Universal Robots PolyScope program: PlaatsenHelicioDemostelling V3.4.1.urp

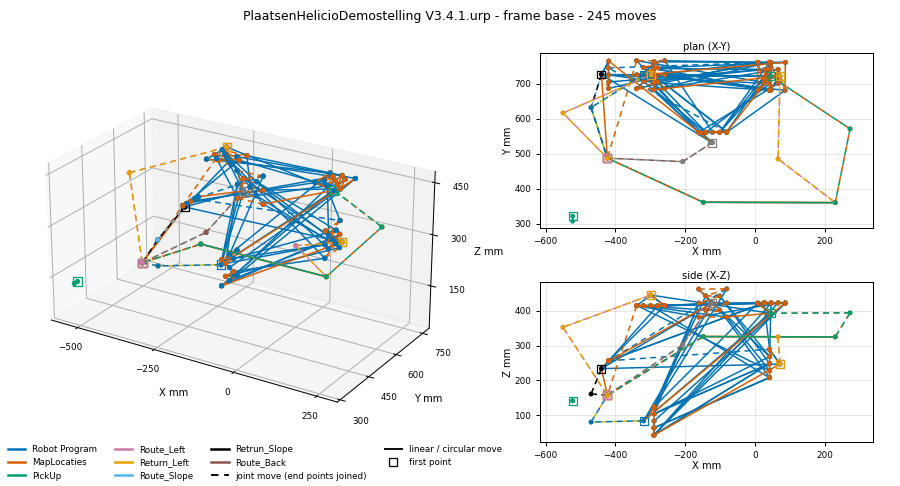
[picture p0: tool path of PlaatsenHelicioDemostelling V3.4.1.urp in frame base, 245 of 246 moves have a stored position in this frame; points joined in program order, loops and branches not executed]
Program PlaatsenHelicioDemostelling V3.4.1 (installation=TestOpstellingVDL directory=/programs/AA VDL ETG FvdT createdIn=5.13.0 lastSavedIn=5.13.0 robotSerialNumber=20195001449)
Calibrated DH parameters: a=[0.000035, -0.365107, -0.323271, 0.000053, -0.00002, 0]; d=[0.181019, -256.633431, 683.600492, -426.792497, 0.119803, 0.115725]; alpha=[1.570596, 0.001914, 0.001103, 1.570723, -1.571951, 0]; deltaTheta=[0, -0.931514, 8.183833, -0.969128, 0.000002, 0]
InitVariablesNode
BeforeStart
  Script file /programs/AA VDL ETG FvdT/Inspectie.script
    | ###
    | # Next functions are for the inspection how deep the helicoils are placed inside their holes ;)
    | # DirectiomalMovement is a variable that will tell the fucntion what axis is used for the movement:
    | # 0: X
    | # 1: Y
    | # 2: Z
    | # 3: XZ
    | ###
    | 
    | 
    | #Arrays to inspect the placed helicoils
    | global arrayStartX        = [0,0,0,0,0,0]
    | global arrayStartZ        = [0,0,0,0,0,0]
    | global arrayFinishX       = [0,0,0,0,0,0]
    | global arrayFinishZ       = [0,0,0,0,0,0]
    | #Results from the inspection
    | global ControlShort      = [0,0,0,0,0,0]
    | global ControlLong       = [0,0,0,0,0,0]
    | global ControlSpecial    = [0,0,0,0,0,0]
    | global ControlWrong      = [0,0,0,0,0,0]
    | global ControlSingle     = [0,0,0,0,0,0]
    | 
    | #How many went wrong while placing helicoils
    | global Interventions     = 0
    | 
    | #When calling this function it will return the wanted XYZ pose from the tcp
    | def Postion(RouteIndex, Start, PostionArrayX,PostionArrayZ):
    |   arrayX = PostionArrayX
    |   arrayZ = PostionArrayZ
    |   freedrive_mode()
    |   sleep(0.01)
    |   Pose  = get_actual_tcp_pose()
    |   end_freedrive_mode()
    |   sleep(0.01)
    |   arrayX[RouteIndex] = Pose[0]
    |   arrayZ[RouteIndex] = Pose[2]
    |   if (Start):
    |     arrayStartX = arrayX
    |     arrayStartZ = arrayZ
    |   else:
    |     arrayFinishX = arrayX
    |     arrayFinishZ = arrayZ
    |   end
    | end
    | 
    | #This function is for checking if the helicoil is placed at the right height everything is in mm. only the postionArrays are in meters
    | # 0: Right
    | # 1: Left
    | # 2: Slope
    | # 3: Back
    | # 4: Flat
    | # 5: Upside
    | def PostionControl(RouteIndex, Side, Route ,ToolcollarDistance, ControlArray):
    | array= ControlArray
    | if Side == 0:
    |   array[RouteIndex] = arrayStartX[RouteIndex] - arrayFinishX[RouteIndex]
    | elif Side == 1:
    |   array[RouteIndex] = arrayStartX[RouteIndex] - arrayFinishX[RouteIndex]
    | elif Side == 2:
    |   xstart = arrayStartX[RouteIndex]/-1
    |   xend = arrayFinishX[RouteIndex]/-1
    |   x = xstart - xend
    |   zstart = arrayStartZ[RouteIndex]
    |   zend   = arrayFinishZ[RouteIndex]
    |   z = zend - zstart
    |   x2 = x*x
    |   z2 = z*z
    |   result= x2+z2
    |   square = sqrt(result)
    |   mmSquare = square * 1000
    |   array[RouteIndex] = mmSquare - 1.5 - ToolcollarDistance
    | elif Side == 3:
    |   array[RouteIndex] = arrayStartX[RouteIndex] - arrayFinishX[RouteIndex]
    | elif Side == 4:
    |   array[RouteIndex] = arrayStartX[RouteIndex] - arrayFinishX[RouteIndex]
    | elif Side == 5:
    |   array[RouteIndex] = arrayStartX[RouteIndex] - arrayFinishX[RouteIndex]
    | end
    | 
    | if Route == 0:
    |   ControlShort = array
    | elif Route == 1:
    |   ControlSpecial = array
    | elif Route == 2:
    |   ControlSingle = array
    | elif Route == 3:
    |   ControlLong = array
    | elif Route == 4:
    |   ControlWrong = array
    | end
    |   if ((array[RouteIndex] < 0.1) and (array[RouteIndex] > 0.3)):
    |     popup("Helicoil outside the correct range of placement", title="Popup", warning=False, error=True)
    |     Interventions = Interventions + 1
    |   end
    | end
  Set DigitalOutput pin=digital_out[6]; digitalValue=1
  bFreedrive := 0
  bIndraaien := 0
  bOppakken := 0
  bUitdraaien := 0
  Route_Index_1 := 0
  URCap Move Shank (OnRobot, OnRobot A/S) dataModel(or-initialized=true, sd-target-pos=0.0)
    'Add conditions here'
Robot Program (runOnlyOnce=false)
  Route_Index_1 := 0
  Wait Condition expression=digital_in[0] or digital_in[1] or digital_in[2] or digital_in[3] or digital_in[4]
  If digital_in[0] and (ChoiceLong≟0)
    Folder LongDemo_1
      SafeHome (positionOptionType=SPEED_AND_ACCELERATION speed=1.047198 acceleration=1.396263 nextMotionTime=2)
      Call PickUp
      Call Route_Left
      MoveL speed 250 mm/s, acceleration 1200 mm/s^2 (useActiveTCP=true) feature=Base
        Waypoint App_Left: TCP in base x=71.596 y=722.403 z=247.152 mm, rx=1.2411 ry=-1.1842 rz=-1.247 rad; joints [84.654, -103.11, -124.444, -129.739, -95.317, 0.645] deg; TCP offset x=153 y=0 z=95.6 mm, rx=0 ry=1.5708 rz=0 rad
      MoveL speed 250 mm/s, acceleration 1200 mm/s^2 (useActiveTCP=true) feature=Center_Left
        Waypoint Left_Hole_1: TCP in base x=41.747 y=681.929 z=288.064 mm, rx=1.241 ry=-1.1844 rz=-1.2467 rad; joints [87.736, -95.501, -128.056, -133.774, -92.257, 0.486] deg; feature pose in base x=41.627 y=722.371 z=247.13 mm, rx=1.2411 ry=-1.1843 rz=-1.2469 rad
      Call ScrewIn_Left
      Call ScrewOut_Left
      Script: PostionControl(Route_Index_1,1, 3,20.4,ControlLong)
      Route_Index_1 := Route_Index_1+1
      MoveL speed 250 mm/s, acceleration 1200 mm/s^2 (useActiveTCP=true) feature=Center_Left
        Waypoint Left_Hole_1: TCP in base x=41.747 y=681.929 z=288.064 mm, rx=1.241 ry=-1.1844 rz=-1.2467 rad; joints [87.736, -95.501, -128.056, -133.774, -92.257, 0.486] deg
      MoveL speed 250 mm/s, acceleration 1200 mm/s^2 (useActiveTCP=true) feature=Base
        Waypoint App_Left: TCP in base x=71.596 y=722.403 z=247.152 mm, rx=1.2411 ry=-1.1842 rz=-1.247 rad; joints [84.654, -103.11, -124.444, -129.739, -95.317, 0.645] deg
      Call Return_Left
      Call PickUp
      Call Route_Slope
      MoveL speed 250 mm/s, acceleration 1200 mm/s^2 (useActiveTCP=true) feature=Base
        Waypoint App_Slope: TCP in base x=-439.97 y=727.052 z=233.948 mm, rx=-1.2131 ry=0.0047 rz=-2.8458 rad; joints [144.347, -130.504, -80.638, -95.321, 64.034, 60.975] deg
      MoveL speed 250 mm/s, acceleration 1200 mm/s^2 (useActiveTCP=true) feature=Center_Slope
        Waypoint Slope_Hole_1: TCP in base x=-418.988 y=765.455 z=256.032 mm, rx=-1.2134 ry=0.0048 rz=-2.8459 rad; joints [141.834, -130.588, -78.129, -96.713, 62.566, 58.706] deg; feature pose in base x=-417.692 y=727.543 z=255.471 mm, rx=-1.2135 ry=0.0049 rz=-2.8456 rad
      Call ScrewIn_Slope
      Call ScrewOut_Slope
      Script: PostionControl(Route_Index_1,2, 3,20.4,ControlLong)
      Route_Index_1 := Route_Index_1+1
      MoveL speed 250 mm/s, acceleration 1200 mm/s^2 (useActiveTCP=true) feature=Center_Slope
        Waypoint Slope_Hole_1: TCP in base x=-418.988 y=765.455 z=256.032 mm, rx=-1.2134 ry=0.0048 rz=-2.8459 rad; joints [141.834, -130.588, -78.129, -96.713, 62.566, 58.706] deg
      MoveL speed 250 mm/s, acceleration 1200 mm/s^2 (useActiveTCP=true) feature=Base
        Waypoint App_Slope: TCP in base x=-439.97 y=727.052 z=233.948 mm, rx=-1.2131 ry=0.0047 rz=-2.8458 rad; joints [144.347, -130.504, -80.638, -95.321, 64.034, 60.975] deg
      Call Retrun_Slope
      Call PickUp
      Call Route_Back
      MoveL speed 250 mm/s, acceleration 1200 mm/s^2 (useActiveTCP=true) feature=Base
        Waypoint App_Back: TCP in base x=-123.1 y=531.725 z=421.395 mm, rx=-1.1912 ry=-1.1756 rz=-1.1726 rad; joints [133.279, -56.474, -130.364, -80.605, 90.835, -48.335] deg
      MoveL speed 250 mm/s, acceleration 1200 mm/s^2 (useActiveTCP=true) feature=Center_Back
        Waypoint Back_Hole_1: TCP in base x=-161.091 y=559.776 z=461.746 mm, rx=-1.1916 ry=-1.1754 rz=-1.1728 rad; joints [134.504, -60.988, -124.308, -82.128, 90.793, -47.089] deg; feature pose in base x=-123.174 y=561.721 z=421.393 mm, rx=-1.1912 ry=-1.1756 rz=-1.1725 rad
      Call ScrewIn_Back
      Call ScrewOut_Back
      Script: PostionControl(Route_Index_1,3, 3,20.4,ControlLong)
      Route_Index_1 := Route_Index_1+1
      MoveL speed 250 mm/s, acceleration 1200 mm/s^2 (useActiveTCP=true) feature=Center_Back
        Waypoint Back_Hole_1: TCP in base x=-161.091 y=559.776 z=461.746 mm, rx=-1.1916 ry=-1.1754 rz=-1.1728 rad; joints [134.504, -60.988, -124.308, -82.128, 90.793, -47.089] deg
      MoveL speed 250 mm/s, acceleration 1200 mm/s^2 (useActiveTCP=true) feature=Base
        Waypoint App_Back: TCP in base x=-123.1 y=531.725 z=421.395 mm, rx=-1.1912 ry=-1.1756 rz=-1.1726 rad; joints [133.279, -56.474, -130.364, -80.605, 90.835, -48.335] deg
      Call Return_Back
      Call PickUp
      Call Route_Right
      MoveL speed 250 mm/s, acceleration 1200 mm/s^2 (useActiveTCP=true) feature=Base
        Waypoint App_Right: TCP in base x=-319.122 y=726.35 z=84.615 mm, rx=-1.8156 ry=0.6848 rz=-1.8051 rad; joints [142.098, -124.495, -115.917, -1.496, 59.13, 44.861] deg; TCP offset x=153 y=0 z=95.6 mm, rx=0 ry=1.5708 rz=0 rad
      MoveL speed 250 mm/s, acceleration 1200 mm/s^2 (useActiveTCP=true) feature=Center_Right
        Waypoint Right_Hole_1: TCP in base x=-288.676 y=762.832 z=123.23 mm, rx=-1.6513 ry=0.8665 rz=-1.6389 rad; joints [140.517, -126.661, -116.023, 15.048, 50.947, 35.529] deg; TCP offset x=153 y=0 z=95.6 mm, rx=0 ry=1.5708 rz=0 rad; feature pose in base x=-289.14 y=726.341 z=83.917 mm, rx=-1.8154 ry=0.6847 rz=-1.8054 rad
      Call ScrewIn_Right
      Call ScrewOut_Right
      Script: PostionControl(Route_Index_1,0, 3,20.4,ControlLong)
      Route_Index_1 := Route_Index_1+1
      MoveL speed 250 mm/s, acceleration 1200 mm/s^2 (useActiveTCP=true) feature=Center_Right
        Waypoint Right_Hole_1: TCP in base x=-288.676 y=762.832 z=123.23 mm, rx=-1.6513 ry=0.8665 rz=-1.6389 rad; joints [140.517, -126.661, -116.023, 15.048, 50.947, 35.529] deg
      MoveL speed 250 mm/s, acceleration 1200 mm/s^2 (useActiveTCP=true) feature=Base
        Waypoint App_Right: TCP in base x=-319.122 y=726.35 z=84.615 mm, rx=-1.8156 ry=0.6848 rz=-1.8051 rad; joints [142.098, -124.495, -115.917, -1.496, 59.13, 44.861] deg; TCP offset x=153 y=0 z=95.6 mm, rx=0 ry=1.5708 rz=0 rad
      Call Retrun_Right
      Call PickUp
      Call Route_Upside
      MoveL speed 250 mm/s, acceleration 1200 mm/s^2 (useActiveTCP=true) feature=Base
        Waypoint App_Upside: TCP in base x=44.432 y=722.092 z=392.585 mm, rx=0.0098 ry=0.0116 rz=-1.5803 rad; joints [105.261, -99.805, -128.74, -130.763, -74.252, 90.052] deg; TCP offset x=153 y=0 z=95.6 mm, rx=0 ry=1.5708 rz=0 rad
      MoveL speed 250 mm/s, acceleration 1200 mm/s^2 (useActiveTCP=true) feature=Base
        Waypoint Upside_Hole_1: TCP in base x=7.793 y=681.564 z=421.754 mm, rx=0.0115 ry=0.0085 rz=-1.1224 rad; joints [99.071, -96.217, -128.805, -134.239, -106.684, 90.097] deg
      Call ScrewIn_Upside
      Call ScrewOut_Upside
      Script: PostionControl(Route_Index_1,5, 3,20.4,ControlLong)
      Route_Index_1 := Route_Index_1+1
      MoveL speed 250 mm/s, acceleration 1200 mm/s^2 (useActiveTCP=true) feature=Base
        Waypoint Upside_Hole_1: TCP in base x=7.793 y=681.564 z=421.754 mm, rx=0.0115 ry=0.0085 rz=-1.1224 rad; joints [99.071, -96.217, -128.805, -134.239, -106.684, 90.097] deg
      MoveL speed 250 mm/s, acceleration 1200 mm/s^2 (useActiveTCP=true) feature=Base
        Waypoint App_Upside: TCP in base x=44.432 y=722.092 z=392.585 mm, rx=0.0098 ry=0.0116 rz=-1.5803 rad; joints [105.261, -99.805, -128.74, -130.763, -74.252, 90.052] deg
      Call Return_Upside
      Call PickUp
      Call Route_Flat
      MoveL speed 250 mm/s, acceleration 1200 mm/s^2 (useActiveTCP=true) feature=Base
        Waypoint App_Flat: TCP in base x=-298.667 y=726.067 z=444.64 mm, rx=-0.093 ry=3.1337 rz=-0.0054 rad; joints [137.032, -122.864, -79.694, 22.109, -43.59, 90.001] deg
      MoveL speed 250 mm/s, acceleration 1200 mm/s^2 (useActiveTCP=true) feature=Center_Flat
        Waypoint Flat_Hole_1: TCP in base x=-259.128 y=686.324 z=414.438 mm, rx=-0.0932 ry=3.1334 rz=-0.006 rad; joints [137.195, -119.277, -88.838, 27.642, -43.744, 89.991] deg; feature pose in base x=-298.69 y=726.112 z=414.639 mm, rx=-0.0931 ry=3.1338 rz=-0.0052 rad
      Call ScrewIn_Flat
      Call ScrewOut_Flat
      Script: PostionControl(Route_Index_1,4, 3,20.4,ControlLong)
      Route_Index_1 := Route_Index_1+1
      MoveL speed 250 mm/s, acceleration 1200 mm/s^2 (useActiveTCP=true) feature=Center_Flat
        Waypoint Flat_Hole_1: TCP in base x=-259.128 y=686.324 z=414.438 mm, rx=-0.0932 ry=3.1334 rz=-0.006 rad; joints [137.195, -119.277, -88.838, 27.642, -43.744, 89.991] deg
      MoveL speed 250 mm/s, acceleration 1200 mm/s^2 (useActiveTCP=true) feature=Base
        Waypoint App_Flat: TCP in base x=-298.667 y=726.067 z=444.64 mm, rx=-0.093 ry=3.1337 rz=-0.0054 rad; joints [137.032, -122.864, -79.694, 22.109, -43.59, 90.001] deg
      Call Return_Flat
      ChoiceLong := ChoiceLong+1
  ElseIf digital_in[0] and (ChoiceLong>1)
    Set DigitalOutput pin=digital_out[2]; digitalValue=1
    Wait Sleep waitTime=0.5
    Wait DigitalInput pin=digital_in[0]; digitalValue=1
    Set DigitalOutput pin=digital_out[2]; digitalValue=0
    Wait Sleep waitTime=0.5
  ElseIf digital_in[0] and (ChoiceLong≟1)
    Folder LongDemo2
      SafeHome (positionOptionType=SPEED_AND_ACCELERATION speed=1.047198 acceleration=1.396263 nextMotionTime=2)
      Call PickUp
      Call Route_Flat
      MoveL speed 250 mm/s, acceleration 1200 mm/s^2 (useActiveTCP=true) feature=Center_Flat
        Waypoint Flat_Hole_2: TCP in base x=-339.559 y=686.213 z=413.913 mm, rx=-0.0931 ry=3.1333 rz=-0.0061 rad; joints [140.84, -123.458, -82.105, 25.101, -47.4, 89.95] deg; feature pose in base x=-298.69 y=726.112 z=414.639 mm, rx=-0.0931 ry=3.1338 rz=-0.0052 rad
      Call ScrewIn_Flat
      Call ScrewOut_Flat
      Script: PostionControl(Route_Index_1,4, 3,20.4,ControlLong)
      Route_Index_1 := Route_Index_1+1
      MoveL speed 250 mm/s, acceleration 1200 mm/s^2 (useActiveTCP=true) feature=Center_Flat
        Waypoint Flat_Hole_2: TCP in base x=-339.559 y=686.213 z=413.913 mm, rx=-0.0931 ry=3.1333 rz=-0.0061 rad; joints [140.84, -123.458, -82.105, 25.101, -47.4, 89.95] deg
      Call Return_Flat
      Call PickUp
      Call Route_Upside
      MoveL speed 250 mm/s, acceleration 1200 mm/s^2 (useActiveTCP=true) feature=Base
        Waypoint Upside_Hole_2: TCP in base x=7.992 y=762.089 z=421.467 mm, rx=0.0114 ry=0.0085 rz=-1.1226 rad; joints [97.734, -103.064, -120.286, -135.906, -108.002, 90.119] deg
      Call ScrewIn_Upside
      Call ScrewOut_Upside
      Script: PostionControl(Route_Index_1,5, 3,20.4,ControlLong)
      Route_Index_1 := Route_Index_1+1
      MoveL speed 250 mm/s, acceleration 1200 mm/s^2 (useActiveTCP=true) feature=Base
        Waypoint Upside_Hole_2: TCP in base x=7.992 y=762.089 z=421.467 mm, rx=0.0114 ry=0.0085 rz=-1.1226 rad; joints [97.734, -103.064, -120.286, -135.906, -108.002, 90.119] deg
      Call Return_Upside
      Call PickUp
      Call Route_Right
      MoveL speed 250 mm/s, acceleration 1200 mm/s^2 (useActiveTCP=true) feature=Center_Right
        Waypoint Right_Hole_2: TCP in base x=-288.899 y=724.109 z=124.718 mm, rx=-1.8156 ry=0.6847 rz=-1.8052 rad; joints [140.747, -119.909, -118.016, -3.275, 59.778, 43.466] deg; feature pose in base x=-289.14 y=726.341 z=83.917 mm, rx=-1.8154 ry=0.6847 rz=-1.8054 rad
      Call ScrewIn_Right
      Call ScrewOut_Right
      Script: PostionControl(Route_Index_1,0, 3,20.4,ControlLong)
      Route_Index_1 := Route_Index_1+1
      MoveL speed 250 mm/s, acceleration 1200 mm/s^2 (useActiveTCP=true) feature=Center_Right
        Waypoint Right_Hole_2: TCP in base x=-288.899 y=724.109 z=124.718 mm, rx=-1.8156 ry=0.6847 rz=-1.8052 rad; joints [140.747, -119.909, -118.016, -3.275, 59.778, 43.466] deg
      Call Retrun_Right
      Call PickUp
      Call Route_Back
      MoveL speed 250 mm/s, acceleration 1200 mm/s^2 (useActiveTCP=true) feature=Center_Back
        Waypoint Back_Hole_2: TCP in base x=-81.106 y=561.818 z=462.255 mm, rx=-1.1915 ry=-1.1754 rz=-1.1728 rad; joints [125.05, -58.623, -125.311, -83.64, 91.187, -56.541] deg; feature pose in base x=-123.174 y=561.721 z=421.393 mm, rx=-1.1912 ry=-1.1756 rz=-1.1725 rad
      SuppressedNode
        Call ScrewIn_Back
      SuppressedNode
        Call ScrewOut_Back
      Script: PostionControl(Route_Index_1,3, 3,20.4,ControlLong)
      Route_Index_1 := Route_Index_1+1
      MoveL speed 250 mm/s, acceleration 1200 mm/s^2 (useActiveTCP=true) feature=Center_Back
        Waypoint Back_Hole_2: TCP in base x=-81.106 y=561.818 z=462.255 mm, rx=-1.1915 ry=-1.1754 rz=-1.1728 rad; joints [125.05, -58.623, -125.311, -83.64, 91.187, -56.541] deg
      Call Return_Back
      Call PickUp
      Call Route_Slope
      MoveJ speed 60 deg/s, acceleration 80 deg/s^2 (useActiveTCP=true) feature=Center_Slope
        Waypoint Slope_Hole_2: TCP in base x=-420.147 y=745.777 z=256.244 mm, rx=-1.2132 ry=0.0049 rz=-2.8457 rad; joints [142.781, -129.419, -80.121, -96.284, 63.105, 59.566] deg; feature pose in base x=-417.692 y=727.543 z=255.471 mm, rx=-1.2135 ry=0.0049 rz=-2.8456 rad
      Call ScrewIn_Slope
      Call ScrewOut_Slope
      Script: PostionControl(Route_Index_1,5, 3,20.4,ControlLong)
      Route_Index_1 := Route_Index_1+1
      MoveJ speed 60 deg/s, acceleration 80 deg/s^2 (useActiveTCP=true) feature=Center_Slope
        Waypoint Slope_Hole_2: TCP in base x=-420.147 y=745.777 z=256.244 mm, rx=-1.2132 ry=0.0049 rz=-2.8457 rad; joints [142.781, -129.419, -80.121, -96.284, 63.105, 59.566] deg
      Call Retrun_Slope
      Call PickUp
      Call Route_Left
      MoveJ speed 60 deg/s, acceleration 80 deg/s^2 (useActiveTCP=true) feature=Center_Left
        Waypoint Left_hole_2: TCP in base x=41.851 y=761.933 z=289.563 mm, rx=1.241 ry=-1.1846 rz=-1.2468 rad; joints [88.048, -101.94, -119.992, -135.397, -91.927, 0.472] deg; feature pose in base x=41.627 y=722.371 z=247.13 mm, rx=1.2411 ry=-1.1843 rz=-1.2469 rad
      Call ScrewIn_Left
      Call ScrewOut_Left
      Script: PostionControl(Route_Index_1,1, 3,20.4,ControlLong)
      Route_Index_1 := Route_Index_1+1
      MoveJ speed 60 deg/s, acceleration 80 deg/s^2 (useActiveTCP=true) feature=Center_Left
        Waypoint Left_hole_2: TCP in base x=41.851 y=761.933 z=289.563 mm, rx=1.241 ry=-1.1846 rz=-1.2468 rad; joints [88.048, -101.94, -119.992, -135.397, -91.927, 0.472] deg
      Call Return_Left
      ChoiceLong := ChoiceLong+1
  If digital_in[2] and (ChoiceSpecial≟0)
    Folder SpacialDemo_1
      SafeHome (positionOptionType=SPEED_AND_ACCELERATION speed=1.047198 acceleration=1.396263 nextMotionTime=2)
      Call PickUp
      Call Route_Upside
      MoveL speed 250 mm/s, acceleration 1200 mm/s^2 (useActiveTCP=true) feature=Base
        Waypoint Upside_Hole_3: TCP in base x=25.312 y=701.594 z=422.409 mm, rx=0.0095 ry=0.0108 rz=-1.6026 rad; joints [108.748, -95.233, -129.852, -134.263, -69.496, 89.993] deg
      Call ScrewIn_Upside
      Call ScrewOut_Upside
      Script: PostionControl(Route_Index_1,5, 1,20.4,ControlSpecial)
      Route_Index_1 := Route_Index_1+1
      MoveL speed 250 mm/s, acceleration 1200 mm/s^2 (useActiveTCP=true) feature=Base
        Waypoint Upside_Hole_3: TCP in base x=25.312 y=701.594 z=422.409 mm, rx=0.0095 ry=0.0108 rz=-1.6026 rad; joints [108.748, -95.233, -129.852, -134.263, -69.496, 89.993] deg
      Call Return_Upside
      Call PickUp
      Call Route_Slope
      MoveL speed 250 mm/s, acceleration 1200 mm/s^2 (useActiveTCP=true) feature=Center_Slope
        Waypoint Slope_Hole_3: TCP in base x=-419.505 y=725.856 z=255.958 mm, rx=-1.2131 ry=0.0047 rz=-2.8457 rad; joints [143.7, -128.19, -82.264, -95.747, 63.645, 60.388] deg; feature pose in base x=-417.692 y=727.543 z=255.471 mm, rx=-1.2135 ry=0.0049 rz=-2.8456 rad
      Call ScrewIn_Slope
      Call ScrewOut_Slope
      Script: PostionControl(Route_Index_1,2, 1,20.4,ControlSpecial)
      Route_Index_1 := Route_Index_1+1
      MoveL speed 250 mm/s, acceleration 1200 mm/s^2 (useActiveTCP=true) feature=Center_Slope
        Waypoint Slope_Hole_3: TCP in base x=-419.505 y=725.856 z=255.958 mm, rx=-1.2131 ry=0.0047 rz=-2.8457 rad; joints [143.7, -128.19, -82.264, -95.747, 63.645, 60.388] deg
      Call Retrun_Slope
      Call PickUp
      Call Route_Flat
      MoveL speed 250 mm/s, acceleration 1200 mm/s^2 (useActiveTCP=true) feature=Center_Flat
        Waypoint Flat_Hole_3: TCP in base x=-279.053 y=706.316 z=414.093 mm, rx=-0.093 ry=3.1333 rz=-0.0061 rad; joints [137.112, -121.662, -85.035, 26.213, -43.671, 89.995] deg; feature pose in base x=-298.69 y=726.112 z=414.639 mm, rx=-0.0931 ry=3.1338 rz=-0.0052 rad
      Call ScrewIn_Flat
      Call ScrewOut_Left
      Script: PostionControl(Route_Index_1,1, 1,20.4,ControlSpecial)
      Route_Index_1 := Route_Index_1+1
      MoveL speed 250 mm/s, acceleration 1200 mm/s^2 (useActiveTCP=true) feature=Center_Flat
        Waypoint Flat_Hole_3: TCP in base x=-279.053 y=706.316 z=414.093 mm, rx=-0.093 ry=3.1333 rz=-0.0061 rad; joints [137.112, -121.662, -85.035, 26.213, -43.671, 89.995] deg
      Call Return_Flat
      ChoiceSpecial := ChoiceSpecial+1
  ElseIf digital_in[2] and (ChoiceSpecial≟1)
    Folder SpacialDemo_2
      SafeHome (positionOptionType=SPEED_AND_ACCELERATION speed=1.047198 acceleration=1.396263 nextMotionTime=2)
      Call PickUp
      Call Route_Flat
      MoveL speed 250 mm/s, acceleration 1200 mm/s^2 (useActiveTCP=true) feature=Center_Flat
        Waypoint Flat_Hole_4: TCP in base x=-319.374 y=706.548 z=413.961 mm, rx=-0.093 ry=3.1333 rz=-0.0061 rad; joints [138.927, -123.752, -81.611, 24.894, -45.487, 89.973] deg
      Call ScrewIn_Flat
      Call ScrewOut_Flat
      Script: PostionControl(Route_Index_1,4, 1,20.4,ControlSpecial)
      Route_Index_1 := Route_Index_1+1
      MoveL speed 250 mm/s, acceleration 1200 mm/s^2 (useActiveTCP=true) feature=Center_Flat
        Waypoint Flat_Hole_4: TCP in base x=-319.374 y=706.548 z=413.961 mm, rx=-0.093 ry=3.1333 rz=-0.0061 rad; joints [138.927, -123.752, -81.611, 24.894, -45.487, 89.973] deg
      Call Return_Flat
      Call PickUp
      Call Route_Upside
      MoveL speed 250 mm/s, acceleration 1200 mm/s^2 (useActiveTCP=true) feature=Base
        Waypoint Upside_Hole_4: TCP in base x=28.457 y=741.552 z=422.373 mm, rx=0.0116 ry=0.0086 rz=-1.1224 rad; joints [95.855, -101.646, -122.034, -135.547, -109.894, 90.144] deg
      Call ScrewIn_Upside
      Call ScrewOut_Upside
      Script: PostionControl(Route_Index_1,5, 1,20.4,ControlSpecial)
      Route_Index_1 := Route_Index_1+1
      MoveL speed 250 mm/s, acceleration 1200 mm/s^2 (useActiveTCP=true) feature=Base
        Waypoint Upside_Hole_4: TCP in base x=28.457 y=741.552 z=422.373 mm, rx=0.0116 ry=0.0086 rz=-1.1224 rad; joints [95.855, -101.646, -122.034, -135.547, -109.894, 90.144] deg
      Call Return_Upside
      Call PickUp
      Call Route_Slope
      MoveL speed 250 mm/s, acceleration 1200 mm/s^2 (useActiveTCP=true) feature=Center_Slope
        Waypoint Slope_Hole_4: TCP in base x=-418.797 y=705.709 z=257.194 mm, rx=-1.2136 ry=0.005 rz=-2.8455 rad; joints [144.651, -126.896, -84.317, -95.345, 64.216, 61.241] deg; feature pose in base x=-417.692 y=727.543 z=255.471 mm, rx=-1.2135 ry=0.0049 rz=-2.8456 rad
      Call ScrewIn_Slope
      Call ScrewOut_Slope
      Script: PostionControl(Route_Index_1,2, 1,20.4,ControlSpecial)
      Route_Index_1 := Route_Index_1+1
      MoveL speed 250 mm/s, acceleration 1200 mm/s^2 (useActiveTCP=true) feature=Center_Slope
        Waypoint Slope_Hole_4: TCP in base x=-418.797 y=705.709 z=257.194 mm, rx=-1.2136 ry=0.005 rz=-2.8455 rad; joints [144.651, -126.896, -84.317, -95.345, 64.216, 61.241] deg
      Call Retrun_Slope
      ChoiceSpecial := ChoiceSpecial+1
  ElseIf digital_in[2] and (ChoiceSpecial≟2)
    Folder SpacialDemo_3
      SafeHome (positionOptionType=SPEED_AND_ACCELERATION speed=1.047198 acceleration=1.396263 nextMotionTime=2)
      Call PickUp
      Call Route_Slope
      MoveL speed 250 mm/s, acceleration 1200 mm/s^2 (useActiveTCP=true) feature=Center_Slope
        Waypoint Slope_Hole_5: TCP in base x=-419.08 y=686.879 z=256.503 mm, rx=-1.2131 ry=0.0048 rz=-2.8457 rad; joints [145.6, -125.867, -86.129, -94.947, 64.778, 62.084] deg
      Call ScrewIn_Slope
      Call ScrewOut_Slope
      Script: PostionControl(Route_Index_1,2, 1,20.4,ControlSpecial)
      Route_Index_1 := Route_Index_1+1
      MoveL speed 250 mm/s, acceleration 1200 mm/s^2 (useActiveTCP=true) feature=Center_Slope
        Waypoint Slope_Hole_5: TCP in base x=-419.08 y=686.879 z=256.503 mm, rx=-1.2131 ry=0.0048 rz=-2.8457 rad; joints [145.6, -125.867, -86.129, -94.947, 64.778, 62.084] deg
      Call Retrun_Slope
      Call PickUp
      Call Route_Flat
      MoveL speed 250 mm/s, acceleration 1200 mm/s^2 (useActiveTCP=true) feature=Center_Flat
        Waypoint Flat_Hole_5: TCP in base x=-258.651 y=725.987 z=414.388 mm, rx=-0.0931 ry=3.1336 rz=-0.0055 rad; joints [135.168, -122.05, -84.362, 25.942, -41.726, 90.022] deg; feature pose in base x=-298.69 y=726.112 z=414.639 mm, rx=-0.0931 ry=3.1338 rz=-0.0052 rad
      Call ScrewIn_Flat
      Call ScrewOut_Flat
      Script: PostionControl(Route_Index_1,4, 1,20.4,ControlSpecial)
      Route_Index_1 := Route_Index_1+1
      MoveL speed 250 mm/s, acceleration 1200 mm/s^2 (useActiveTCP=true) feature=Center_Flat
        Waypoint Flat_Hole_5: TCP in base x=-258.651 y=725.987 z=414.388 mm, rx=-0.0931 ry=3.1336 rz=-0.0055 rad; joints [135.168, -122.05, -84.362, 25.942, -41.726, 90.022] deg
      Call Return_Flat
      Call PickUp
      Call Route_Upside
      MoveL speed 250 mm/s, acceleration 1200 mm/s^2 (useActiveTCP=true) feature=Base
        Waypoint Upside_Hole_5: TCP in base x=45.602 y=681.858 z=421.646 mm, rx=0.0094 ry=0.0108 rz=-1.5922 rad; joints [106.795, -93.58, -131.803, -133.972, -72.048, 90.021] deg
      SuppressedNode
        Call ScrewIn_Upside
      SuppressedNode
        Call ScrewOut_Upside
      Script: PostionControl(Route_Index_1,4, 1,20.5,ControlSpecial)
      MoveL speed 250 mm/s, acceleration 1200 mm/s^2 (useActiveTCP=true) feature=Base
        Waypoint Upside_Hole_5: TCP in base x=45.602 y=681.858 z=421.646 mm, rx=0.0094 ry=0.0108 rz=-1.5922 rad; joints [106.795, -93.58, -131.803, -133.972, -72.048, 90.021] deg
      Call Return_Upside
      ChoiceSpecial := ChoiceSpecial+1
  If digital_in[3] and (ChoiceWrong≟0)
    Folder WrongDemo_1
      SafeHome (positionOptionType=SPEED_AND_ACCELERATION speed=1.047198 acceleration=1.396263 nextMotionTime=2)
      Call PickUp
      Call Route_Left
      MoveL speed 250 mm/s, acceleration 1200 mm/s^2 (useActiveTCP=true) feature=Center_Left
        Waypoint Left_Hole_3: TCP in base x=41.78 y=700.693 z=268.277 mm, rx=1.2407 ry=-1.1848 rz=-1.2467 rad; joints [87.825, -98.689, -127.06, -131.593, -92.143, 0.481] deg; feature pose in base x=41.627 y=722.371 z=247.13 mm, rx=1.2411 ry=-1.1843 rz=-1.2469 rad
      Call ScrewIn_Left
      Call ScrewOut_Left
      Script: PostionControl(Route_Index_1,1, 4,20.4,ControlWrong)
      Route_Index_1 := Route_Index_1+1
      MoveL speed 250 mm/s, acceleration 1200 mm/s^2 (useActiveTCP=true) feature=Center_Left
        Waypoint Left_Hole_3: TCP in base x=41.78 y=700.693 z=268.277 mm, rx=1.2407 ry=-1.1848 rz=-1.2467 rad; joints [87.825, -98.689, -127.06, -131.593, -92.143, 0.481] deg
      Call Return_Left
      Call PickUp
      Call Route_Back
      MoveL speed 250 mm/s, acceleration 1200 mm/s^2 (useActiveTCP=true) feature=Center_Back
        Waypoint Back_Hole_3: TCP in base x=-141.317 y=560.737 z=442.316 mm, rx=-1.1916 ry=-1.1753 rz=-1.1725 rad; joints [132.279, -60.529, -126.481, -80.438, 90.901, -49.317] deg; feature pose in base x=-123.174 y=561.721 z=421.393 mm, rx=-1.1912 ry=-1.1756 rz=-1.1725 rad
      Call ScrewIn_Back
      Call ScrewOut_Back
      Script: PostionControl(Route_Index_1,1, 3,20.4,ControlWrong)
      Route_Index_1 := Route_Index_1+1
      MoveL speed 250 mm/s, acceleration 1200 mm/s^2 (useActiveTCP=true) feature=Center_Back
        Waypoint Back_Hole_3: TCP in base x=-141.317 y=560.737 z=442.316 mm, rx=-1.1916 ry=-1.1753 rz=-1.1725 rad; joints [132.279, -60.529, -126.481, -80.438, 90.901, -49.317] deg
      Call Return_Back
      Call PickUp
      Call Route_Right
      MoveL speed 250 mm/s, acceleration 1200 mm/s^2 (useActiveTCP=true) feature=Center_Right
        Waypoint Right_Hole_3: TCP in base x=-289.204 y=683.885 z=123.717 mm, rx=-1.8156 ry=0.6847 rz=-1.8051 rad; joints [143.374, -117.868, -121.795, -2.924, 58.544, 46.159] deg; feature pose in base x=-289.14 y=726.341 z=83.917 mm, rx=-1.8154 ry=0.6847 rz=-1.8054 rad
      Call ScrewIn_Right
      Call ScrewOut_Right
      Script: PostionControl(Route_Index_1,0, 4,20.4,ControlWrong)
      Route_Index_1 := Route_Index_1+1
      MoveL speed 250 mm/s, acceleration 1200 mm/s^2 (useActiveTCP=true) feature=Center_Right
        Waypoint Right_Hole_3: TCP in base x=-289.204 y=683.885 z=123.717 mm, rx=-1.8156 ry=0.6847 rz=-1.8051 rad; joints [143.374, -117.868, -121.795, -2.924, 58.544, 46.159] deg
      Call Retrun_Right
    ChoiceWrong := ChoiceWrong+1
  ElseIf digital_in[3] and (ChoiceWrong≟2)
    Folder WrongDemo_3
      SafeHome (positionOptionType=SPEED_AND_ACCELERATION speed=1.047198 acceleration=1.396263 nextMotionTime=2)
      Call PickUp
      Call Route_Back
      MoveL speed 250 mm/s, acceleration 1200 mm/s^2 (useActiveTCP=true) feature=Center_Back
        Waypoint Back_Hole_5: TCP in base x=-160.808 y=560.703 z=421.755 mm, rx=-1.1913 ry=-1.1757 rz=-1.1725 rad; joints [134.374, -61.689, -128.015, -77.73, 90.806, -47.239] deg; feature pose in base x=-123.174 y=561.721 z=421.393 mm, rx=-1.1912 ry=-1.1756 rz=-1.1725 rad
      Call ScrewIn_Back
      Call ScrewOut_Back
      Script: PostionControl(Route_Index_1,3, 4,20.4,ControlWrong)
      Route_Index_1 := Route_Index_1+1
      MoveL speed 250 mm/s, acceleration 1200 mm/s^2 (useActiveTCP=true) feature=Center_Back
        Waypoint Back_Hole_5: TCP in base x=-160.808 y=560.703 z=421.755 mm, rx=-1.1913 ry=-1.1757 rz=-1.1725 rad; joints [134.374, -61.689, -128.015, -77.73, 90.806, -47.239] deg
      Call Return_Back
      Call PickUp
      Call Route_Right
      MoveL speed 250 mm/s, acceleration 1200 mm/s^2 (useActiveTCP=true) feature=Center_Right
        Waypoint Right_Hole_5: TCP in base x=-289.172 y=703.708 z=104.449 mm, rx=-1.8156 ry=0.6847 rz=-1.8052 rad; joints [142.057, -120.721, -120.085, -1.08, 59.155, 44.81] deg; feature pose in base x=-289.14 y=726.341 z=83.917 mm, rx=-1.8154 ry=0.6847 rz=-1.8054 rad
      Call ScrewIn_Right
      Call ScrewOut_Right
      Script: PostionControl(Route_Index_1,0, 4,20.4,ControlWrong)
      Route_Index_1 := Route_Index_1+1
      MoveL speed 250 mm/s, acceleration 1200 mm/s^2 (useActiveTCP=true) feature=Center_Right
        Waypoint Right_Hole_5: TCP in base x=-289.172 y=703.708 z=104.449 mm, rx=-1.8156 ry=0.6847 rz=-1.8052 rad; joints [142.057, -120.721, -120.085, -1.08, 59.155, 44.81] deg
      Call Retrun_Right
      Call PickUp
      Call Route_Left
      MoveL speed 250 mm/s, acceleration 1200 mm/s^2 (useActiveTCP=true) feature=Center_Left
        Waypoint Left_Hole_5: TCP in base x=41.621 y=681.741 z=247.936 mm, rx=1.2407 ry=-1.1848 rz=-1.2466 rad; joints [87.758, -98.951, -129.738, -128.658, -92.209, 0.483] deg; feature pose in base x=41.627 y=722.371 z=247.13 mm, rx=1.2411 ry=-1.1843 rz=-1.2469 rad
      Call ScrewIn_Left
      Call ScrewOut_Left
      Script: PostionControl(Route_Index_1,1, 4,20.4,ControlWrong)
      Route_Index_1 := Route_Index_1+1
      MoveL speed 250 mm/s, acceleration 1200 mm/s^2 (useActiveTCP=true) feature=Center_Left
        Waypoint Left_Hole_5: TCP in base x=41.621 y=681.741 z=247.936 mm, rx=1.2407 ry=-1.1848 rz=-1.2466 rad; joints [87.758, -98.951, -129.738, -128.658, -92.209, 0.483] deg
      Call Return_Left
    ChoiceWrong := ChoiceWrong+1
  ElseIf digital_in[3] and (ChoiceWrong≟1)
    Folder WrongDemo_2
      SafeHome (positionOptionType=SPEED_AND_ACCELERATION speed=1.047198 acceleration=1.396263 nextMotionTime=2)
      Call PickUp
      Call Route_Right
      MoveL speed 250 mm/s, acceleration 1200 mm/s^2 (useActiveTCP=true) feature=Center_Right
        Waypoint Right_Hole_4: TCP in base x=-288.818 y=744.018 z=104.467 mm, rx=-1.8156 ry=0.6845 rz=-1.8053 rad; joints [139.527, -122.763, -116.22, -1.612, 60.368, 42.243] deg; feature pose in base x=-289.14 y=726.341 z=83.917 mm, rx=-1.8154 ry=0.6847 rz=-1.8054 rad
      Call ScrewIn_Right
      Call ScrewOut_Right
      Script: PostionControl(Route_Index_1,0, 4,20.4,ControlWrong)
      Route_Index_1 := Route_Index_1+1
      MoveL speed 250 mm/s, acceleration 1200 mm/s^2 (useActiveTCP=true) feature=Center_Right
        Waypoint Right_Hole_4: TCP in base x=-288.818 y=744.018 z=104.467 mm, rx=-1.8156 ry=0.6845 rz=-1.8053 rad; joints [139.527, -122.763, -116.22, -1.612, 60.368, 42.243] deg
      Call Retrun_Right
      Call PickUp
      Call Route_Left
      MoveL speed 250 mm/s, acceleration 1200 mm/s^2 (useActiveTCP=true) feature=Center_Left
        Waypoint Left_Hole_4: TCP in base x=41.829 y=741.625 z=268.564 mm, rx=1.2407 ry=-1.1848 rz=-1.2468 rad; joints [87.983, -101.916, -122.916, -132.511, -91.98, 0.478] deg; feature pose in base x=41.627 y=722.371 z=247.13 mm, rx=1.2411 ry=-1.1843 rz=-1.2469 rad
      Call ScrewIn_Left
      Call ScrewOut_Left
      Script: PostionControl(Route_Index_1,1, 4,20.4,ControlWrong)
      Route_Index_1 := Route_Index_1+1
      MoveL speed 250 mm/s, acceleration 1200 mm/s^2 (useActiveTCP=true) feature=Center_Left
        Waypoint Left_Hole_4: TCP in base x=41.829 y=741.625 z=268.564 mm, rx=1.2407 ry=-1.1848 rz=-1.2468 rad; joints [87.983, -101.916, -122.916, -132.511, -91.98, 0.478] deg
      Call Return_Left
      Call PickUp
      Call Route_Back
      MoveL speed 250 mm/s, acceleration 1200 mm/s^2 (useActiveTCP=true) feature=Center_Back
        Waypoint Back_Hole_4: TCP in base x=-100.931 y=561.75 z=441.913 mm, rx=-1.1915 ry=-1.1753 rz=-1.1725 rad; joints [127.507, -59.311, -127.065, -81.147, 91.1, -54.089] deg; feature pose in base x=-123.174 y=561.721 z=421.393 mm, rx=-1.1912 ry=-1.1756 rz=-1.1725 rad
      Call ScrewIn_Back
      Call ScrewOut_Back
      Script: PostionControl(Route_Index_1,3, 4,20.4,ControlWrong)
      Route_Index_1 := Route_Index_1+1
      MoveL speed 250 mm/s, acceleration 1200 mm/s^2 (useActiveTCP=true) feature=Center_Back
        Waypoint Back_Hole_4: TCP in base x=-100.931 y=561.75 z=441.913 mm, rx=-1.1915 ry=-1.1753 rz=-1.1725 rad; joints [127.507, -59.311, -127.065, -81.147, 91.1, -54.089] deg
      Call Return_Back
    ChoiceWrong := ChoiceWrong+1
  If digital_in[1] and (ChoiceShort≟0)
    Folder ShortDemo_1
      SafeHome (positionOptionType=SPEED_AND_ACCELERATION speed=1.047198 acceleration=1.396263 nextMotionTime=2)
      Call PickUp
      Call Route_Left
      MoveL speed 250 mm/s, acceleration 1200 mm/s^2 (useActiveTCP=true) feature=Center_Left
        Waypoint Left_Hole_6: TCP in base x=41.661 y=721.943 z=248.573 mm, rx=1.2412 ry=-1.1844 rz=-1.247 rad; joints [87.923, -102.032, -125.679, -129.603, -92.048, 0.482] deg; feature pose in base x=41.627 y=722.371 z=247.13 mm, rx=1.2411 ry=-1.1843 rz=-1.2469 rad
      Call ScrewIn_Left
      Call ScrewOut_Left
      Script: PostionControl(Route_Index_1,1, 0,20.4,ControlShort)
      Route_Index_1 := Route_Index_1+1
      MoveL speed 250 mm/s, acceleration 1200 mm/s^2 (useActiveTCP=true) feature=Center_Left
        Waypoint Left_Hole_6: TCP in base x=41.661 y=721.943 z=248.573 mm, rx=1.2412 ry=-1.1844 rz=-1.247 rad; joints [87.923, -102.032, -125.679, -129.603, -92.048, 0.482] deg
      Call Return_Left
      Call PickUp
      Call Route_Right
      MoveL speed 250 mm/s, acceleration 1200 mm/s^2 (useActiveTCP=true) feature=Center_Right
        Waypoint Right_Hole_10: TCP in base x=-289.595 y=723.359 z=43.588 mm, rx=-1.8156 ry=0.6846 rz=-1.8051 rad; joints [140.827, -127.475, -118.143, 4.367, 59.733, 43.565] deg; feature pose in base x=-289.14 y=726.341 z=83.917 mm, rx=-1.8154 ry=0.6847 rz=-1.8054 rad
      Call ScrewIn_Right
      Call ScrewOut_Right
      Script: PostionControl(Route_Index_1,0, 0,20.4,ControlShort)
      Route_Index_1 := Route_Index_1+1
      MoveL speed 250 mm/s, acceleration 1200 mm/s^2 (useActiveTCP=true) feature=Center_Right
        Waypoint Right_Hole_10: TCP in base x=-289.595 y=723.359 z=43.588 mm, rx=-1.8156 ry=0.6846 rz=-1.8051 rad; joints [140.827, -127.475, -118.143, 4.367, 59.733, 43.565] deg
      Call Retrun_Right
      Call PickUp
      Call Route_Upside
      MoveL speed 250 mm/s, acceleration 1200 mm/s^2 (useActiveTCP=true) feature=Base
        Waypoint Upside_Hole_6: TCP in base x=45.629 y=721.749 z=421.143 mm, rx=0.0098 ry=0.0115 rz=-1.5802 rad; joints [105.13, -97.306, -127.635, -134.374, -74.396, 90.048] deg
      Call ScrewIn_Upside
      Call ScrewOut_Upside
      Script: PostionControl(Route_Index_1,5, 0,20.4,ControlShort)
      Route_Index_1 := Route_Index_1+1
      MoveL speed 250 mm/s, acceleration 1200 mm/s^2 (useActiveTCP=true) feature=Base
        Waypoint Upside_Hole_6: TCP in base x=45.629 y=721.749 z=421.143 mm, rx=0.0098 ry=0.0115 rz=-1.5802 rad; joints [105.13, -97.306, -127.635, -134.374, -74.396, 90.048] deg
      Call Return_Upside
    ChoiceShort := ChoiceShort+1
  ElseIf digital_in[1] and (ChoiceShort≟1)
    Folder ShortDemo_2
      SafeHome (positionOptionType=SPEED_AND_ACCELERATION speed=1.047198 acceleration=1.396263 nextMotionTime=2)
      Call PickUp
      Call Route_Upside
      MoveL speed 250 mm/s, acceleration 1200 mm/s^2 (useActiveTCP=true) feature=Base
        Waypoint Upside_Hole_7: TCP in base x=46.075 y=761.507 z=422.684 mm, rx=0.0095 ry=0.0109 rz=-1.5923 rad; joints [104.212, -100.607, -123.332, -135.408, -74.616, 90.054] deg
      Call ScrewIn_Upside
      Call ScrewOut_Upside
      Script: PostionControl(Route_Index_1,5, 0,20.4,ControlShort)
      Route_Index_1 := Route_Index_1+1
      MoveL speed 250 mm/s, acceleration 1200 mm/s^2 (useActiveTCP=true) feature=Base
        Waypoint Upside_Hole_7: TCP in base x=46.075 y=761.507 z=422.684 mm, rx=0.0095 ry=0.0109 rz=-1.5923 rad; joints [104.212, -100.607, -123.332, -135.408, -74.616, 90.054] deg
      Call Return_Upside
      Call PickUp
      Call Route_Flat
      MoveL speed 250 mm/s, acceleration 1200 mm/s^2 (useActiveTCP=true) feature=Center_Flat
        Waypoint Flat_Hole_10: TCP in base x=-258.485 y=766.369 z=414.023 mm, rx=-0.0934 ry=3.1332 rz=-0.0063 rad; joints [133.268, -125.019, -79.495, 23.998, -39.818, 90.046] deg; feature pose in base x=-298.69 y=726.112 z=414.639 mm, rx=-0.0931 ry=3.1338 rz=-0.0052 rad
      Call ScrewIn_Flat
      Call ScrewOut_Flat
      Script: PostionControl(Route_Index_1,4, 0,20.4,ControlShort)
      Route_Index_1 := Route_Index_1+1
      MoveL speed 250 mm/s, acceleration 1200 mm/s^2 (useActiveTCP=true) feature=Center_Flat
        Waypoint Flat_Hole_10: TCP in base x=-258.485 y=766.369 z=414.023 mm, rx=-0.0934 ry=3.1332 rz=-0.0063 rad; joints [133.268, -125.019, -79.495, 23.998, -39.818, 90.046] deg
      Call Return_Flat
      Call PickUp
      Call Route_Back
      MoveL speed 250 mm/s, acceleration 1200 mm/s^2 (useActiveTCP=true) feature=Center_Back
        Waypoint Back_Hole_6: TCP in base x=-121.665 y=561.713 z=422.253 mm, rx=-1.1913 ry=-1.1757 rz=-1.1725 rad; joints [129.968, -60.258, -128.629, -78.606, 90.991, -51.642] deg; feature pose in base x=-123.174 y=561.721 z=421.393 mm, rx=-1.1912 ry=-1.1756 rz=-1.1725 rad
      Call ScrewIn_Back
      Call ScrewOut_Back
      Script: PostionControl(Route_Index_1,3, 0,20.4,ControlShort)
      Route_Index_1 := Route_Index_1+1
      MoveL speed 250 mm/s, acceleration 1200 mm/s^2 (useActiveTCP=true) feature=Center_Back
        Waypoint Back_Hole_6: TCP in base x=-121.665 y=561.713 z=422.253 mm, rx=-1.1913 ry=-1.1757 rz=-1.1725 rad; joints [129.968, -60.258, -128.629, -78.606, 90.991, -51.642] deg
      Call Return_Back
    ChoiceShort := ChoiceShort+1
  ElseIf digital_in[1] and (ChoiceShort≟2)
    Folder ShortDemo_3
      SafeHome (positionOptionType=SPEED_AND_ACCELERATION speed=1.047198 acceleration=1.396263 nextMotionTime=2)
      Call PickUp
      Call Route_Back
      MoveL speed 250 mm/s, acceleration 1200 mm/s^2 (useActiveTCP=true) feature=Center_Back
        Waypoint Back_Hole_7: TCP in base x=-81.214 y=561.376 z=422.087 mm, rx=-1.1914 ry=-1.1756 rz=-1.1725 rad; joints [125.096, -59.068, -129.167, -79.339, 91.196, -56.509] deg
      Call ScrewIn_Back
      Call ScrewOut_Back
      Script: PostionControl(Route_Index_1,3, 0,20.4,ControlShort)
      Route_Index_1 := Route_Index_1+1
      MoveL speed 250 mm/s, acceleration 1200 mm/s^2 (useActiveTCP=true) feature=Center_Back
        Waypoint Back_Hole_7: TCP in base x=-81.214 y=561.376 z=422.087 mm, rx=-1.1914 ry=-1.1756 rz=-1.1725 rad; joints [125.096, -59.068, -129.167, -79.339, 91.196, -56.509] deg
      Call Return_Back
      Call PickUp
      Call Route_Upside
      MoveL speed 250 mm/s, acceleration 1200 mm/s^2 (useActiveTCP=true) feature=Base
        Waypoint Upside_Hole_10: TCP in base x=85.909 y=681.545 z=420.624 mm, rx=0.0097 ry=0.0115 rz=-1.58 rad; joints [101.434, -94.182, -131.306, -133.827, -78.105, 90.095] deg
      Call ScrewIn_Upside
      Call ScrewOut_Upside
      Script: PostionControl(Route_Index_1,5, 0,20.4,ControlShort)
      Route_Index_1 := Route_Index_1+1
      MoveL speed 250 mm/s, acceleration 1200 mm/s^2 (useActiveTCP=true) feature=Base
        Waypoint Upside_Hole_10: TCP in base x=85.909 y=681.545 z=420.624 mm, rx=0.0097 ry=0.0115 rz=-1.58 rad; joints [101.434, -94.182, -131.306, -133.827, -78.105, 90.095] deg
      Call Return_Upside
      Call PickUp
      Call Route_Right
      MoveL speed 250 mm/s, acceleration 1200 mm/s^2 (useActiveTCP=true) feature=Center_Right
        Waypoint Right_Hole_6: TCP in base x=-289.189 y=724.036 z=83.936 mm, rx=-1.8154 ry=0.6846 rz=-1.8053 rad; joints [140.767, -123.659, -118.205, 0.642, 59.757, 43.494] deg; feature pose in base x=-289.14 y=726.341 z=83.917 mm, rx=-1.8154 ry=0.6847 rz=-1.8054 rad
      Call ScrewIn_Right
      Call ScrewOut_Right
      Script: PostionControl(Route_Index_1,0, 0,20.4,ControlShort)
      Route_Index_1 := Route_Index_1+1
      MoveL speed 250 mm/s, acceleration 1200 mm/s^2 (useActiveTCP=true) feature=Center_Right
        Waypoint Right_Hole_6: TCP in base x=-289.189 y=724.036 z=83.936 mm, rx=-1.8154 ry=0.6846 rz=-1.8053 rad; joints [140.767, -123.659, -118.205, 0.642, 59.757, 43.494] deg
      Call Retrun_Right
    ChoiceShort := ChoiceShort+1
  ElseIf digital_in[1] and (ChoiceShort≟3)
    Folder ShortDemo_4
      SafeHome (positionOptionType=SPEED_AND_ACCELERATION speed=1.047198 acceleration=1.396263 nextMotionTime=2)
      Call PickUp
      Call Route_Right
      MoveL speed 250 mm/s, acceleration 1200 mm/s^2 (useActiveTCP=true) feature=Center_Right
        Waypoint Right_Hole_7: TCP in base x=-289.188 y=743.625 z=64.091 mm, rx=-1.8156 ry=0.6847 rz=-1.8052 rad; joints [139.569, -126.432, -116.277, 2.096, 60.342, 42.295] deg
      Call ScrewIn_Right
      Call ScrewOut_Right
      Wait Sleep waitTime=10
      SuppressedNode
        Script: PostionControl(Route_Index_1,0, 0,20.4,ControlShort)
      Route_Index_1 := Route_Index_1+1
      MoveL speed 250 mm/s, acceleration 1200 mm/s^2 (useActiveTCP=true) feature=Center_Right
        Waypoint Right_Hole_7: TCP in base x=-289.188 y=743.625 z=64.091 mm, rx=-1.8156 ry=0.6847 rz=-1.8052 rad; joints [139.569, -126.432, -116.277, 2.096, 60.342, 42.295] deg
      Call Retrun_Right
      Call PickUp
      Call Route_Left
      MoveL speed 250 mm/s, acceleration 1200 mm/s^2 (useActiveTCP=true) feature=Center_Left
        Waypoint Left_Hole_10: TCP in base x=41.475 y=682.374 z=207.743 mm, rx=1.2403 ry=-1.1849 rz=-1.2465 rad; joints [87.783, -102.844, -131.026, -123.494, -92.168, 0.493] deg; feature pose in base x=41.627 y=722.371 z=247.13 mm, rx=1.2411 ry=-1.1843 rz=-1.2469 rad
      Call ScrewIn_Left
      Call ScrewOut_Left
      Script: PostionControl(Route_Index_1,1, 0,20.4,ControlShort)
      Route_Index_1 := Route_Index_1+1
      MoveL speed 250 mm/s, acceleration 1200 mm/s^2 (useActiveTCP=true) feature=Center_Left
        Waypoint Left_Hole_10: TCP in base x=41.475 y=682.374 z=207.743 mm, rx=1.2403 ry=-1.1849 rz=-1.2465 rad; joints [87.783, -102.844, -131.026, -123.494, -92.168, 0.493] deg
      Call Return_Left
      Call PickUp
      Call Route_Flat
      MoveL speed 250 mm/s, acceleration 1200 mm/s^2 (useActiveTCP=true) feature=Center_Flat
        Waypoint Flat_Hole_6: TCP in base x=-298.708 y=726.085 z=414.645 mm, rx=-0.0931 ry=3.1337 rz=-0.0053 rad; joints [137.035, -124.015, -81.089, 24.659, -43.595, 90] deg; feature pose in base x=-298.69 y=726.112 z=414.639 mm, rx=-0.0931 ry=3.1338 rz=-0.0052 rad
      Call ScrewIn_Flat
      Wait Sleep waitTime=1
      Call ScrewOut_Flat
      Wait Sleep waitTime=20
      Script: PostionControl(Route_Index_1,4, 0,20.4,ControlShort)
      Route_Index_1 := Route_Index_1+1
      MoveL speed 250 mm/s, acceleration 1200 mm/s^2 (useActiveTCP=true) feature=Center_Flat
        Waypoint Flat_Hole_6: TCP in base x=-298.708 y=726.085 z=414.645 mm, rx=-0.0931 ry=3.1337 rz=-0.0053 rad; joints [137.035, -124.015, -81.089, 24.659, -43.595, 90] deg
      Call Return_Flat
    ChoiceShort := ChoiceShort+1
  ElseIf digital_in[1] and (ChoiceShort≟4)
    Folder ShortDemo_5
      SafeHome (positionOptionType=SPEED_AND_ACCELERATION speed=1.047198 acceleration=1.396263 nextMotionTime=2)
      Call PickUp
      Call Route_Flat
      MoveL speed 250 mm/s, acceleration 1200 mm/s^2 (useActiveTCP=true) feature=Center_Flat
        Waypoint Flat_Hole_7: TCP in base x=-338.996 y=726.099 z=413.978 mm, rx=-0.093 ry=3.1337 rz=-0.0056 rad; joints [138.802, -126.174, -77.546, 23.276, -45.368, 89.975] deg
      Call ScrewIn_Flat
      Call ScrewOut_Flat
      Script: PostionControl(Route_Index_1,4, 0,20.4,ControlShort)
      Route_Index_1 := Route_Index_1+1
      MoveL speed 250 mm/s, acceleration 1200 mm/s^2 (useActiveTCP=true) feature=Center_Flat
        Waypoint Flat_Hole_7: TCP in base x=-338.996 y=726.099 z=413.978 mm, rx=-0.093 ry=3.1337 rz=-0.0056 rad; joints [138.802, -126.174, -77.546, 23.276, -45.368, 89.975] deg
      Call Return_Flat
      Call PickUp
      Call Route_Back
      MoveL speed 250 mm/s, acceleration 1200 mm/s^2 (useActiveTCP=true) feature=Center_Back
        Waypoint Back_Hole_10: TCP in base x=-160.783 y=561.693 z=381.7 mm, rx=-1.1914 ry=-1.1755 rz=-1.1727 rad; joints [134.278, -62.825, -131.574, -73.029, 90.813, -47.316] deg; feature pose in base x=-123.174 y=561.721 z=421.393 mm, rx=-1.1912 ry=-1.1756 rz=-1.1725 rad
      Call ScrewIn_Back
      Call ScrewOut_Back
      Script: PostionControl(Route_Index_1,3, 0,20.4,ControlShort)
      Route_Index_1 := Route_Index_1+1
      MoveL speed 250 mm/s, acceleration 1200 mm/s^2 (useActiveTCP=true) feature=Center_Back
        Waypoint Back_Hole_10: TCP in base x=-160.783 y=561.693 z=381.7 mm, rx=-1.1914 ry=-1.1755 rz=-1.1727 rad; joints [134.278, -62.825, -131.574, -73.029, 90.813, -47.316] deg
      Call Return_Back
      Call PickUp
      Call Route_Upside
      MoveL speed 250 mm/s, acceleration 1200 mm/s^2 (useActiveTCP=true) feature=Base
        Waypoint Upside_Hole_8: TCP in base x=65.869 y=701.366 z=421.757 mm, rx=0.0095 ry=0.011 rz=-1.6027 rad; joints [103.929, -95.564, -129.571, -134.21, -74.311, 90.056] deg
      Call ScrewIn_Upside
      Call ScrewOut_Upside
      Script: PostionControl(Route_Index_1,5, 0,20.4,ControlShort)
      Route_Index_1 := Route_Index_1+1
      MoveL speed 250 mm/s, acceleration 1200 mm/s^2 (useActiveTCP=true) feature=Base
        Waypoint Upside_Hole_8: TCP in base x=65.869 y=701.366 z=421.757 mm, rx=0.0095 ry=0.011 rz=-1.6027 rad; joints [103.929, -95.564, -129.571, -134.21, -74.311, 90.056] deg
      Call Return_Upside
    ChoiceShort := ChoiceShort+1
  ElseIf digital_in[1] and (ChoiceShort≟5)
    Folder ShortDemo_6
      SafeHome (positionOptionType=SPEED_AND_ACCELERATION speed=1.047198 acceleration=1.396263 nextMotionTime=2)
      Call PickUp
      Call Route_Upside
      MoveL speed 250 mm/s, acceleration 1200 mm/s^2 (useActiveTCP=true) feature=Base
        Waypoint Upside_Hole_9: TCP in base x=66.109 y=741.352 z=422.584 mm, rx=0.0095 ry=0.0108 rz=-1.6026 rad; joints [102.804, -99.034, -125.314, -135.007, -75.433, 90.067] deg
      Call ScrewIn_Upside
      Call ScrewOut_Upside
      Script: PostionControl(Route_Index_1,5, 0,20.4,ControlShort)
      Route_Index_1 := Route_Index_1+1
      MoveL speed 250 mm/s, acceleration 1200 mm/s^2 (useActiveTCP=true) feature=Base
        Waypoint Upside_Hole_9: TCP in base x=66.109 y=741.352 z=422.584 mm, rx=0.0095 ry=0.0108 rz=-1.6026 rad; joints [102.804, -99.034, -125.314, -135.007, -75.433, 90.067] deg
      Call Return_Upside
      Call PickUp
      Call Route_Right
      MoveL speed 250 mm/s, acceleration 1200 mm/s^2 (useActiveTCP=true) feature=Center_Right
        Waypoint Right_Hole_11: TCP in base x=-289.905 y=683.248 z=43.271 mm, rx=-1.8157 ry=0.6845 rz=-1.8052 rad; joints [143.448, -125.804, -121.937, 5.097, 58.506, 46.262] deg; feature pose in base x=-289.14 y=726.341 z=83.917 mm, rx=-1.8154 ry=0.6847 rz=-1.8054 rad
      Call ScrewIn_Right
      Call ScrewOut_Right
      Script: PostionControl(Route_Index_1,0, 0,20.4,ControlShort)
      Route_Index_1 := Route_Index_1+1
      MoveL speed 250 mm/s, acceleration 1200 mm/s^2 (useActiveTCP=true) feature=Center_Right
        Waypoint Right_Hole_11: TCP in base x=-289.905 y=683.248 z=43.271 mm, rx=-1.8157 ry=0.6845 rz=-1.8052 rad; joints [143.448, -125.804, -121.937, 5.097, 58.506, 46.262] deg
      Call Retrun_Right
      Call PickUp
      Call Route_Left
      MoveL speed 250 mm/s, acceleration 1200 mm/s^2 (useActiveTCP=true) feature=Center_Left
        Waypoint Left_Hole_7: TCP in base x=41.655 y=761.751 z=248.951 mm, rx=1.2409 ry=-1.1844 rz=-1.2466 rad; joints [88.067, -105.009, -121.541, -130.787, -91.907, 0.479] deg; feature pose in base x=41.627 y=722.371 z=247.13 mm, rx=1.2411 ry=-1.1843 rz=-1.2469 rad
      Call ScrewIn_Left
      Call ScrewOut_Left
      Script: PostionControl(Route_Index_1,1, 0,20.4,ControlShort)
      Route_Index_1 := Route_Index_1+1
      MoveL speed 250 mm/s, acceleration 1200 mm/s^2 (useActiveTCP=true) feature=Center_Left
        Waypoint Left_Hole_7: TCP in base x=41.655 y=761.751 z=248.951 mm, rx=1.2409 ry=-1.1844 rz=-1.2466 rad; joints [88.067, -105.009, -121.541, -130.787, -91.907, 0.479] deg
      Call Return_Left
    ChoiceShort := ChoiceShort+1
  ElseIf digital_in[1] and (ChoiceShort≟6)
    Folder ShortDemo_7
      SafeHome (positionOptionType=SPEED_AND_ACCELERATION speed=1.047198 acceleration=1.396263 nextMotionTime=2)
      Call PickUp
      Call Route_Left
      MoveL speed 250 mm/s, acceleration 1200 mm/s^2 (useActiveTCP=true) feature=Center_Left
        Waypoint Left_Hole_8: TCP in base x=41.551 y=701.515 z=228.336 mm, rx=1.2406 ry=-1.1849 rz=-1.2464 rad; joints [87.856, -102.268, -128.442, -126.647, -92.104, 0.476] deg
      Call ScrewIn_Left
      Call ScrewOut_Left
      Script: PostionControl(Route_Index_1,1, 0,20.4,ControlShort)
      Route_Index_1 := Route_Index_1+1
      MoveL speed 250 mm/s, acceleration 1200 mm/s^2 (useActiveTCP=true) feature=Center_Left
        Waypoint Left_Hole_8: TCP in base x=41.551 y=701.515 z=228.336 mm, rx=1.2406 ry=-1.1849 rz=-1.2464 rad; joints [87.856, -102.268, -128.442, -126.647, -92.104, 0.476] deg
      Call Return_Left
      Call PickUp
      Call Route_Flat
      MoveL speed 250 mm/s, acceleration 1200 mm/s^2 (useActiveTCP=true) feature=Center_Flat
        Waypoint Flat_Hole_11: TCP in base x=-339.071 y=766.535 z=415.174 mm, rx=-0.0929 ry=3.1332 rz=-0.0061 rad; joints [136.895, -129.083, -72.456, 21.043, -43.467, 90.009] deg; feature pose in base x=-298.69 y=726.112 z=414.639 mm, rx=-0.0931 ry=3.1338 rz=-0.0052 rad
      Call ScrewIn_Flat
      Call ScrewOut_Flat
      Script: PostionControl(Route_Index_1,4, 0,20.4,ControlShort)
      Route_Index_1 := Route_Index_1+1
      MoveL speed 250 mm/s, acceleration 1200 mm/s^2 (useActiveTCP=true) feature=Center_Flat
        Waypoint Flat_Hole_11: TCP in base x=-339.071 y=766.535 z=415.174 mm, rx=-0.0929 ry=3.1332 rz=-0.0061 rad; joints [136.895, -129.083, -72.456, 21.043, -43.467, 90.009] deg
      Call Return_Flat
      Call PickUp
      Call Route_Back
      MoveL speed 250 mm/s, acceleration 1200 mm/s^2 (useActiveTCP=true) feature=Center_Back
        Waypoint Back_Hole_8: TCP in base x=-140.676 y=561.721 z=401.738 mm, rx=-1.1916 ry=-1.1757 rz=-1.1725 rad; joints [132.111, -61.411, -130.184, -75.873, 90.912, -49.489] deg; feature pose in base x=-123.174 y=561.721 z=421.393 mm, rx=-1.1912 ry=-1.1756 rz=-1.1725 rad
      Call ScrewIn_Back
      Call ScrewOut_Back
      Script: PostionControl(Route_Index_1,3, 0,20.4,ControlShort)
      Route_Index_1 := Route_Index_1+1
      MoveL speed 250 mm/s, acceleration 1200 mm/s^2 (useActiveTCP=true) feature=Center_Back
        Waypoint Back_Hole_8: TCP in base x=-140.676 y=561.721 z=401.738 mm, rx=-1.1916 ry=-1.1757 rz=-1.1725 rad; joints [132.111, -61.411, -130.184, -75.873, 90.912, -49.489] deg
      Call Return_Back
    ChoiceShort := ChoiceShort+1
  ElseIf digital_in[1] and (ChoiceShort≟7)
    Folder ShortDemo_8
      SafeHome (positionOptionType=SPEED_AND_ACCELERATION speed=1.047198 acceleration=1.396263 nextMotionTime=2)
      Call PickUp
      Call Route_Back
      MoveL speed 250 mm/s, acceleration 1200 mm/s^2 (useActiveTCP=true) feature=Center_Back
        Waypoint Back_Hole_9: TCP in base x=-101.153 y=561.292 z=401.897 mm, rx=-1.1916 ry=-1.1756 rz=-1.1724 rad; joints [127.575, -59.981, -130.818, -76.737, 91.107, -54.022] deg
      Call ScrewIn_Back
      Call ScrewOut_Back
      Script: PostionControl(Route_Index_1,3, 0,20.4,ControlShort)
      Route_Index_1 := Route_Index_1+1
      MoveL speed 250 mm/s, acceleration 1200 mm/s^2 (useActiveTCP=true) feature=Center_Back
        Waypoint Back_Hole_9: TCP in base x=-101.153 y=561.292 z=401.897 mm, rx=-1.1916 ry=-1.1756 rz=-1.1724 rad; joints [127.575, -59.981, -130.818, -76.737, 91.107, -54.022] deg
      Call Return_Back
      Call PickUp
      Call Route_Left
      MoveL speed 250 mm/s, acceleration 1200 mm/s^2 (useActiveTCP=true) feature=Center_Left
        Waypoint Left_Hole_11: TCP in base x=41.584 y=762.28 z=209.041 mm, rx=1.2405 ry=-1.1851 rz=-1.2466 rad; joints [88.087, -108.35, -122.704, -126.306, -91.852, 0.471] deg; feature pose in base x=41.627 y=722.371 z=247.13 mm, rx=1.2411 ry=-1.1843 rz=-1.2469 rad
      Call ScrewIn_Left
      Call ScrewOut_Left
      Script: PostionControl(Route_Index_1,1, 0,20.4,ControlShort)
      Route_Index_1 := Route_Index_1+1
      MoveL speed 250 mm/s, acceleration 1200 mm/s^2 (useActiveTCP=true) feature=Center_Left
        Waypoint Left_Hole_11: TCP in base x=41.584 y=762.28 z=209.041 mm, rx=1.2405 ry=-1.1851 rz=-1.2466 rad; joints [88.087, -108.35, -122.704, -126.306, -91.852, 0.471] deg
      Call Return_Left
      Call PickUp
      Call Route_Right
      MoveL speed 250 mm/s, acceleration 1200 mm/s^2 (useActiveTCP=true) feature=Center_Right
        Waypoint Right_Hole_8: TCP in base x=-289.54 y=703.581 z=64.622 mm, rx=-1.8157 ry=0.6846 rz=-1.8052 rad; joints [142.083, -124.553, -120.133, 2.778, 59.14, 44.847] deg; feature pose in base x=-289.14 y=726.341 z=83.917 mm, rx=-1.8154 ry=0.6847 rz=-1.8054 rad
      Call ScrewIn_Right
      Call ScrewOut_Right
      Script: PostionControl(Route_Index_1,0, 0,20.4,ControlShort)
      Route_Index_1 := Route_Index_1+1
      MoveL speed 250 mm/s, acceleration 1200 mm/s^2 (useActiveTCP=true) feature=Center_Right
        Waypoint Right_Hole_8: TCP in base x=-289.54 y=703.581 z=64.622 mm, rx=-1.8157 ry=0.6846 rz=-1.8052 rad; joints [142.083, -124.553, -120.133, 2.778, 59.14, 44.847] deg
      Call Retrun_Right
    ChoiceShort := ChoiceShort+1
  ElseIf digital_in[1] and (ChoiceShort≟8)
    Folder ShortDemo_9
      SafeHome (positionOptionType=SPEED_AND_ACCELERATION speed=1.047198 acceleration=1.396263 nextMotionTime=2)
      Call PickUp
      Call Route_Right
      MoveL speed 250 mm/s, acceleration 1200 mm/s^2 (useActiveTCP=true) feature=Center_Right
        Waypoint Right_Hole_9: TCP in base x=-289.208 y=763.273 z=44.061 mm, rx=-1.8155 ry=0.6845 rz=-1.8054 rad; joints [138.417, -129.173, -114.225, 3.341, 60.906, 41.149] deg
      Call ScrewIn_Right
      Call ScrewOut_Right
      Script: PostionControl(Route_Index_1,0, 0,20.4,ControlShort)
      Route_Index_1 := Route_Index_1+1
      MoveL speed 250 mm/s, acceleration 1200 mm/s^2 (useActiveTCP=true) feature=Center_Right
        Waypoint Right_Hole_9: TCP in base x=-289.208 y=763.273 z=44.061 mm, rx=-1.8155 ry=0.6845 rz=-1.8054 rad; joints [138.417, -129.173, -114.225, 3.341, 60.906, 41.149] deg
      Call Retrun_Right
      Call PickUp
      Call Route_Upside
      MoveL speed 250 mm/s, acceleration 1200 mm/s^2 (useActiveTCP=true) feature=Base
        Waypoint Upside_Hole_11: TCP in base x=86.561 y=761.692 z=422.63 mm, rx=0.0095 ry=0.011 rz=-1.5797 rad; joints [99.629, -101.038, -122.79, -135.513, -79.917, 90.119] deg
      Call ScrewIn_Upside
      Call ScrewOut_Upside
      Script: PostionControl(Route_Index_1,5, 0,20.4,ControlShort)
      Route_Index_1 := Route_Index_1+1
      MoveL speed 250 mm/s, acceleration 1200 mm/s^2 (useActiveTCP=true) feature=Base
        Waypoint Upside_Hole_11: TCP in base x=86.561 y=761.692 z=422.63 mm, rx=0.0095 ry=0.011 rz=-1.5797 rad; joints [99.629, -101.038, -122.79, -135.513, -79.917, 90.119] deg
      Call Return_Upside
      Call PickUp
      Call Route_Flat
      MoveL speed 250 mm/s, acceleration 1200 mm/s^2 (useActiveTCP=true) feature=Center_Flat
        Waypoint Flat_Hole_8: TCP in base x=-278.546 y=746.2 z=413.871 mm, rx=-0.0933 ry=3.133 rz=-0.0065 rad; joints [135.145, -124.496, -80.39, 24.372, -41.696, 90.021] deg; feature pose in base x=-298.69 y=726.112 z=414.639 mm, rx=-0.0931 ry=3.1338 rz=-0.0052 rad
      Call ScrewIn_Flat
      Call ScrewOut_Flat
      Script: PostionControl(Route_Index_1,4, 0,20.4,ControlShort)
      Route_Index_1 := Route_Index_1+1
      MoveL speed 250 mm/s, acceleration 1200 mm/s^2 (useActiveTCP=true) feature=Center_Flat
        Waypoint Flat_Hole_8: TCP in base x=-278.546 y=746.2 z=413.871 mm, rx=-0.0933 ry=3.133 rz=-0.0065 rad; joints [135.145, -124.496, -80.39, 24.372, -41.696, 90.021] deg
      Call Return_Flat
    ChoiceShort := ChoiceShort+1
  ElseIf digital_in[1] and (ChoiceShort≟9)
    Folder ShortDemo_10
      SafeHome (positionOptionType=SPEED_AND_ACCELERATION speed=1.047198 acceleration=1.396263 nextMotionTime=2)
      Call PickUp
      Call Route_Flat
      MoveL speed 250 mm/s, acceleration 1200 mm/s^2 (useActiveTCP=true) feature=Center_Flat
        Waypoint Flat_Hole_9: TCP in base x=-319.133 y=746.557 z=413.724 mm, rx=-0.0931 ry=3.1332 rz=-0.0062 rad; joints [136.962, -126.589, -76.881, 22.979, -43.523, 89.999] deg
      Call ScrewIn_Flat
      Call ScrewOut_Flat
      Script: PostionControl(Route_Index_1,4, 0,20.4,ControlShort)
      Route_Index_1 := Route_Index_1+1
      MoveL speed 250 mm/s, acceleration 1200 mm/s^2 (useActiveTCP=true) feature=Center_Flat
        Waypoint Flat_Hole_9: TCP in base x=-319.133 y=746.557 z=413.724 mm, rx=-0.0931 ry=3.1332 rz=-0.0062 rad; joints [136.962, -126.589, -76.881, 22.979, -43.523, 89.999] deg
      Call Return_Flat
      Call PickUp
      Call Route_Back
      MoveL speed 250 mm/s, acceleration 1200 mm/s^2 (useActiveTCP=true) feature=Center_Back
        Waypoint Back_Hole_11: TCP in base x=-81.177 y=562.223 z=381.762 mm, rx=-1.1914 ry=-1.1753 rz=-1.1727 rad; joints [125.024, -60.093, -132.831, -74.643, 91.199, -56.566] deg; feature pose in base x=-123.174 y=561.721 z=421.393 mm, rx=-1.1912 ry=-1.1756 rz=-1.1725 rad
      Call ScrewIn_Back
      Call ScrewOut_Back
      Script: PostionControl(Route_Index_1,3, 0,20.4,ControlShort)
      Route_Index_1 := Route_Index_1+1
      MoveL speed 250 mm/s, acceleration 1200 mm/s^2 (useActiveTCP=true) feature=Center_Back
        Waypoint Back_Hole_11: TCP in base x=-81.177 y=562.223 z=381.762 mm, rx=-1.1914 ry=-1.1753 rz=-1.1727 rad; joints [125.024, -60.093, -132.831, -74.643, 91.199, -56.566] deg
      Call Return_Back
      Call PickUp
      Call Route_Left
      MoveL speed 250 mm/s, acceleration 1200 mm/s^2 (useActiveTCP=true) feature=Center_Left
        Waypoint Left_Hole_9: TCP in base x=41.634 y=742.006 z=228.723 mm, rx=1.2408 ry=-1.1848 rz=-1.2467 rad; joints [88.007, -105.221, -124.269, -127.852, -91.948, 0.477] deg; feature pose in base x=41.627 y=722.371 z=247.13 mm, rx=1.2411 ry=-1.1843 rz=-1.2469 rad
      Call ScrewIn_Left
      Call ScrewOut_Left
      Script: PostionControl(Route_Index_1,1, 0,20.4,ControlShort)
      Route_Index_1 := Route_Index_1+1
      MoveL speed 250 mm/s, acceleration 1200 mm/s^2 (useActiveTCP=true) feature=Center_Left
        Waypoint Left_Hole_9: TCP in base x=41.634 y=742.006 z=228.723 mm, rx=1.2408 ry=-1.1848 rz=-1.2467 rad; joints [88.007, -105.221, -124.269, -127.852, -91.948, 0.477] deg
      Call Return_Left
    ChoiceShort := ChoiceShort+1
SubProgram -> Route_Upside
SubProgram -> Return_Upside
SubProgram -> Route_Left
SubProgram -> Return_Left
SubProgram -> Route_Back
SubProgram -> Return_Back
SubProgram -> Route_Flat
SubProgram -> Return_Flat
SubProgram -> Route_Slope
SubProgram -> Retrun_Slope
SubProgram -> Route_Right
SubProgram -> Retrun_Right
SubProgram -> PickUp
SubProgram -> ScrewOut_Upside
SubProgram -> ScrewOut_Back
SubProgram -> ScrewOut_Left
SubProgram -> ScrewOut_Flat
SubProgram -> ScrewOut_Right
SubProgram -> ScrewOut_Slope
SubProgram -> ScrewIn_Upside
SubProgram -> ScrewIn_Right
SubProgram -> ScrewIn_Back
SubProgram -> ScrewIn_Left
SubProgram -> ScrewIn_Slope
SubProgram -> ScrewIn_Flat
Event  expression=bIndraaien
  Script: sd_tighten(0,30,1,0)
Event  expression=bOppakken
  Script: sd_tighten(0,30,3,0)
Event  expression=bUitdraaien
  Script: sd_loosen(2,30,0)
SubProgram MapLocaties (keepSynchronizedWithDisk=false)
  Folder Holes
    MoveJ speed 60 deg/s, acceleration 80 deg/s^2 (useActiveTCP=true) feature=Base
      Waypoint App_Flat: TCP in base x=-298.667 y=726.067 z=444.64 mm, rx=-0.093 ry=3.1337 rz=-0.0054 rad; joints [137.032, -122.864, -79.694, 22.109, -43.59, 90.001] deg
    MoveJ speed 60 deg/s, acceleration 80 deg/s^2 (useActiveTCP=true) feature=Center_Flat
      Waypoint Flat_Hole_1: motionParameters(jointSpeed=1.047198 jointAcceleration=1.396263 cartesianSpeed=0.25 cartesianAcceleration=1.2); TCP in base x=-259.128 y=686.324 z=414.438 mm, rx=-0.0932 ry=3.1334 rz=-0.006 rad; joints [137.195, -119.277, -88.838, 27.642, -43.744, 89.991] deg; feature pose in base x=-298.69 y=726.112 z=414.639 mm, rx=-0.0931 ry=3.1338 rz=-0.0052 rad
      Waypoint Flat_Hole_2: TCP in base x=-339.559 y=686.213 z=413.913 mm, rx=-0.0931 ry=3.1333 rz=-0.0061 rad; joints [140.84, -123.458, -82.105, 25.101, -47.4, 89.95] deg
      Waypoint Flat_Hole_3: TCP in base x=-279.053 y=706.316 z=414.093 mm, rx=-0.093 ry=3.1333 rz=-0.0061 rad; joints [137.112, -121.662, -85.035, 26.213, -43.671, 89.995] deg
      Waypoint Flat_Hole_4: TCP in base x=-319.374 y=706.548 z=413.961 mm, rx=-0.093 ry=3.1333 rz=-0.0061 rad; joints [138.927, -123.752, -81.611, 24.894, -45.487, 89.973] deg
      Waypoint Flat_Hole_5: TCP in base x=-258.651 y=725.987 z=414.388 mm, rx=-0.0931 ry=3.1336 rz=-0.0055 rad; joints [135.168, -122.05, -84.362, 25.942, -41.726, 90.022] deg
      Waypoint Flat_Hole_6: TCP in base x=-298.708 y=726.085 z=414.645 mm, rx=-0.0931 ry=3.1337 rz=-0.0053 rad; joints [137.035, -124.015, -81.089, 24.659, -43.595, 90] deg; feature pose in base x=-298.69 y=726.112 z=414.639 mm, rx=-0.0931 ry=3.1338 rz=-0.0052 rad
      Waypoint Flat_Hole_7: TCP in base x=-338.996 y=726.099 z=413.978 mm, rx=-0.093 ry=3.1337 rz=-0.0056 rad; joints [138.802, -126.174, -77.546, 23.276, -45.368, 89.975] deg; feature pose in base x=-298.69 y=726.112 z=414.639 mm, rx=-0.0931 ry=3.1338 rz=-0.0052 rad
      Waypoint Flat_Hole_8: TCP in base x=-278.546 y=746.2 z=413.871 mm, rx=-0.0933 ry=3.133 rz=-0.0065 rad; joints [135.145, -124.496, -80.39, 24.372, -41.696, 90.021] deg; feature pose in base x=-298.69 y=726.112 z=414.639 mm, rx=-0.0931 ry=3.1338 rz=-0.0052 rad
      Waypoint Flat_Hole_9: TCP in base x=-319.133 y=746.557 z=413.724 mm, rx=-0.0931 ry=3.1332 rz=-0.0062 rad; joints [136.962, -126.589, -76.881, 22.979, -43.523, 89.999] deg; feature pose in base x=-298.69 y=726.112 z=414.639 mm, rx=-0.0931 ry=3.1338 rz=-0.0052 rad
      Waypoint Flat_Hole_10: TCP in base x=-258.485 y=766.369 z=414.023 mm, rx=-0.0934 ry=3.1332 rz=-0.0063 rad; joints [133.268, -125.019, -79.495, 23.998, -39.818, 90.046] deg
      Waypoint Flat_Hole_11: TCP in base x=-339.071 y=766.535 z=415.174 mm, rx=-0.0929 ry=3.1332 rz=-0.0061 rad; joints [136.895, -129.083, -72.456, 21.043, -43.467, 90.009] deg
  MoveJ speed 60 deg/s, acceleration 80 deg/s^2 (useActiveTCP=true) feature=Base
    Waypoint Start_Home: TCP in base x=-422.908 y=487.357 z=157.584 mm, rx=-3.0115 ry=0.7424 rz=0.0187 rad; joints [144.514, -115.165, -138.926, 75.412, 97.807, 88.299] deg
  MoveL speed 250 mm/s, acceleration 1200 mm/s^2 (useActiveTCP=true) feature=Base
    Waypoint App_Slope: TCP in base x=-439.97 y=727.052 z=233.948 mm, rx=-1.2131 ry=0.0047 rz=-2.8458 rad; joints [144.347, -130.504, -80.638, -95.321, 64.034, 60.975] deg
  MoveJ speed 60 deg/s, acceleration 80 deg/s^2 (useActiveTCP=true) feature=Center_Slope
    Waypoint Slope_Hole_5: TCP in base x=-419.08 y=686.879 z=256.503 mm, rx=-1.2131 ry=0.0048 rz=-2.8457 rad; joints [145.6, -125.867, -86.129, -94.947, 64.778, 62.084] deg; feature pose in base x=-417.692 y=727.543 z=255.471 mm, rx=-1.2135 ry=0.0049 rz=-2.8456 rad
    Waypoint Slope_Hole_4: TCP in base x=-418.797 y=705.709 z=257.194 mm, rx=-1.2136 ry=0.005 rz=-2.8455 rad; joints [144.651, -126.896, -84.317, -95.345, 64.216, 61.241] deg
    Waypoint Slope_Hole_3: motionParameters(jointSpeed=1.047198 jointAcceleration=1.396263 cartesianSpeed=0.25 cartesianAcceleration=1.2); TCP in base x=-419.505 y=725.856 z=255.958 mm, rx=-1.2131 ry=0.0047 rz=-2.8457 rad; joints [143.7, -128.19, -82.264, -95.747, 63.645, 60.388] deg
    Waypoint Slope_Hole_2: TCP in base x=-420.147 y=745.777 z=256.244 mm, rx=-1.2132 ry=0.0049 rz=-2.8457 rad; joints [142.781, -129.419, -80.121, -96.284, 63.105, 59.566] deg
    Waypoint Slope_Hole_1: motionParameters(jointSpeed=1.047198 jointAcceleration=1.396263 cartesianSpeed=0.25 cartesianAcceleration=1.2); TCP in base x=-418.988 y=765.455 z=256.032 mm, rx=-1.2134 ry=0.0048 rz=-2.8459 rad; joints [141.834, -130.588, -78.129, -96.713, 62.566, 58.706] deg
  MoveL speed 250 mm/s, acceleration 1200 mm/s^2 (useActiveTCP=true) feature=Base
    Waypoint App_Back: TCP in base x=-123.1 y=531.725 z=421.395 mm, rx=-1.1912 ry=-1.1756 rz=-1.1726 rad; joints [133.279, -56.474, -130.364, -80.605, 90.835, -48.335] deg
  MoveJ speed 60 deg/s, acceleration 80 deg/s^2 (useActiveTCP=true) feature=Center_Back
    Waypoint Back_Hole_1: TCP in base x=-161.091 y=559.776 z=461.746 mm, rx=-1.1916 ry=-1.1754 rz=-1.1728 rad; joints [134.504, -60.988, -124.308, -82.128, 90.793, -47.089] deg; feature pose in base x=-123.174 y=561.721 z=421.393 mm, rx=-1.1912 ry=-1.1756 rz=-1.1725 rad
    Waypoint Back_Hole_2: TCP in base x=-81.106 y=561.818 z=462.255 mm, rx=-1.1915 ry=-1.1754 rz=-1.1728 rad; joints [125.05, -58.623, -125.311, -83.64, 91.187, -56.541] deg
    Waypoint Back_Hole_3: TCP in base x=-141.317 y=560.737 z=442.316 mm, rx=-1.1916 ry=-1.1753 rz=-1.1725 rad; joints [132.279, -60.529, -126.481, -80.438, 90.901, -49.317] deg
    Waypoint Back_Hole_4: TCP in base x=-100.931 y=561.75 z=441.913 mm, rx=-1.1915 ry=-1.1753 rz=-1.1725 rad; joints [127.507, -59.311, -127.065, -81.147, 91.1, -54.089] deg
    Waypoint Back_Hole_5: TCP in base x=-160.808 y=560.703 z=421.755 mm, rx=-1.1913 ry=-1.1757 rz=-1.1725 rad; joints [134.374, -61.689, -128.015, -77.73, 90.806, -47.239] deg
    Waypoint Back_Hole_6: TCP in base x=-121.665 y=561.713 z=422.253 mm, rx=-1.1913 ry=-1.1757 rz=-1.1725 rad; joints [129.968, -60.258, -128.629, -78.606, 90.991, -51.642] deg
    Waypoint Back_Hole_7: TCP in base x=-81.214 y=561.376 z=422.087 mm, rx=-1.1914 ry=-1.1756 rz=-1.1725 rad; joints [125.096, -59.068, -129.167, -79.339, 91.196, -56.509] deg
    Waypoint Back_Hole_8: TCP in base x=-140.676 y=561.721 z=401.738 mm, rx=-1.1916 ry=-1.1757 rz=-1.1725 rad; joints [132.111, -61.411, -130.184, -75.873, 90.912, -49.489] deg
    Waypoint Back_Hole_9: TCP in base x=-101.153 y=561.292 z=401.897 mm, rx=-1.1916 ry=-1.1756 rz=-1.1724 rad; joints [127.575, -59.981, -130.818, -76.737, 91.107, -54.022] deg
    Waypoint Back_Hole_10: TCP in base x=-160.783 y=561.693 z=381.7 mm, rx=-1.1914 ry=-1.1755 rz=-1.1727 rad; joints [134.278, -62.825, -131.574, -73.029, 90.813, -47.316] deg
    Waypoint Back_Hole_11: TCP in base x=-81.177 y=562.223 z=381.762 mm, rx=-1.1914 ry=-1.1753 rz=-1.1727 rad; joints [125.024, -60.093, -132.831, -74.643, 91.199, -56.566] deg
  MoveL speed 250 mm/s, acceleration 1200 mm/s^2 (useActiveTCP=true) feature=Base
    Waypoint App_Upside: TCP in base x=44.432 y=722.092 z=392.585 mm, rx=0.0098 ry=0.0116 rz=-1.5803 rad; joints [105.261, -99.805, -128.74, -130.763, -74.252, 90.052] deg
  MoveL speed 250 mm/s, acceleration 1200 mm/s^2 (useActiveTCP=true) feature=Base
    Waypoint Upside_Hole_1: TCP in base x=7.793 y=681.564 z=421.754 mm, rx=0.0115 ry=0.0085 rz=-1.1224 rad; joints [99.071, -96.217, -128.805, -134.239, -106.684, 90.097] deg
    Waypoint Upside_Hole_2: TCP in base x=7.992 y=762.089 z=421.467 mm, rx=0.0114 ry=0.0085 rz=-1.1226 rad; joints [97.734, -103.064, -120.286, -135.906, -108.002, 90.119] deg
    Waypoint Upside_Hole_3: TCP in base x=25.312 y=701.594 z=422.409 mm, rx=0.0095 ry=0.0108 rz=-1.6026 rad; joints [108.748, -95.233, -129.852, -134.263, -69.496, 89.993] deg
    Waypoint Upside_Hole_4: TCP in base x=28.457 y=741.552 z=422.373 mm, rx=0.0116 ry=0.0086 rz=-1.1224 rad; joints [95.855, -101.646, -122.034, -135.547, -109.894, 90.144] deg
    Waypoint Upside_Hole_5: TCP in base x=45.602 y=681.858 z=421.646 mm, rx=0.0094 ry=0.0108 rz=-1.5922 rad; joints [106.795, -93.58, -131.803, -133.972, -72.048, 90.021] deg
    Waypoint Upside_Hole_6: TCP in base x=45.629 y=721.749 z=421.143 mm, rx=0.0098 ry=0.0115 rz=-1.5802 rad; joints [105.13, -97.306, -127.635, -134.374, -74.396, 90.048] deg
    Waypoint Upside_Hole_7: TCP in base x=46.075 y=761.507 z=422.684 mm, rx=0.0095 ry=0.0109 rz=-1.5923 rad; joints [104.212, -100.607, -123.332, -135.408, -74.616, 90.054] deg
    Waypoint Upside_Hole_8: TCP in base x=65.869 y=701.366 z=421.757 mm, rx=0.0095 ry=0.011 rz=-1.6027 rad; joints [103.929, -95.564, -129.571, -134.21, -74.311, 90.056] deg
    Waypoint Upside_Hole_9: TCP in base x=66.109 y=741.352 z=422.584 mm, rx=0.0095 ry=0.0108 rz=-1.6026 rad; joints [102.804, -99.034, -125.314, -135.007, -75.433, 90.067] deg
    Waypoint Upside_Hole_10: TCP in base x=85.909 y=681.545 z=420.624 mm, rx=0.0097 ry=0.0115 rz=-1.58 rad; joints [101.434, -94.182, -131.306, -133.827, -78.105, 90.095] deg
    Waypoint Upside_Hole_11: TCP in base x=86.561 y=761.692 z=422.63 mm, rx=0.0095 ry=0.011 rz=-1.5797 rad; joints [99.629, -101.038, -122.79, -135.513, -79.917, 90.119] deg
  SuppressedNode
    MoveL speed 250 mm/s, acceleration 1200 mm/s^2 (useActiveTCP=true) feature=Base
      SuppressedNode
        Waypoint App_Flat: TCP in base x=-298.667 y=726.067 z=444.64 mm, rx=-0.093 ry=3.1337 rz=-0.0054 rad; joints [137.032, -122.864, -79.694, 22.109, -43.59, 90.001] deg
  MoveL speed 250 mm/s, acceleration 1200 mm/s^2 (useActiveTCP=true) feature=Base
    Waypoint App_Right: TCP in base x=-319.122 y=726.35 z=84.615 mm, rx=-1.8156 ry=0.6848 rz=-1.8051 rad; joints [142.098, -124.495, -115.917, -1.496, 59.13, 44.861] deg; TCP offset x=153 y=0 z=95.6 mm, rx=0 ry=1.5708 rz=0 rad
  MoveJ speed 60 deg/s, acceleration 80 deg/s^2 (useActiveTCP=true) feature=Center_Right
    Waypoint Right_Hole_1: TCP in base x=-288.676 y=762.832 z=123.23 mm, rx=-1.6513 ry=0.8665 rz=-1.6389 rad; joints [140.517, -126.661, -116.023, 15.048, 50.947, 35.529] deg; TCP offset x=153 y=0 z=95.6 mm, rx=0 ry=1.5708 rz=0 rad; feature pose in base x=-289.14 y=726.341 z=83.917 mm, rx=-1.8154 ry=0.6847 rz=-1.8054 rad
    Waypoint Right_Hole_2: TCP in base x=-288.899 y=724.109 z=124.718 mm, rx=-1.8156 ry=0.6847 rz=-1.8052 rad; joints [140.747, -119.909, -118.016, -3.275, 59.778, 43.466] deg
    Waypoint Right_Hole_3: TCP in base x=-289.204 y=683.885 z=123.717 mm, rx=-1.8156 ry=0.6847 rz=-1.8051 rad; joints [143.374, -117.868, -121.795, -2.924, 58.544, 46.159] deg
    Waypoint Right_Hole_4: TCP in base x=-288.818 y=744.018 z=104.467 mm, rx=-1.8156 ry=0.6845 rz=-1.8053 rad; joints [139.527, -122.763, -116.22, -1.612, 60.368, 42.243] deg
    Waypoint Right_Hole_5: TCP in base x=-289.172 y=703.708 z=104.449 mm, rx=-1.8156 ry=0.6847 rz=-1.8052 rad; joints [142.057, -120.721, -120.085, -1.08, 59.155, 44.81] deg
    Waypoint Right_Hole_6: TCP in base x=-289.189 y=724.036 z=83.936 mm, rx=-1.8154 ry=0.6846 rz=-1.8053 rad; joints [140.767, -123.659, -118.205, 0.642, 59.757, 43.494] deg
    Waypoint Right_Hole_7: TCP in base x=-289.188 y=743.625 z=64.091 mm, rx=-1.8156 ry=0.6847 rz=-1.8052 rad; joints [139.569, -126.432, -116.277, 2.096, 60.342, 42.295] deg
    Waypoint Right_Hole_8: TCP in base x=-289.54 y=703.581 z=64.622 mm, rx=-1.8157 ry=0.6846 rz=-1.8052 rad; joints [142.083, -124.553, -120.133, 2.778, 59.14, 44.847] deg
    Waypoint Right_Hole_9: TCP in base x=-289.208 y=763.273 z=44.061 mm, rx=-1.8155 ry=0.6845 rz=-1.8054 rad; joints [138.417, -129.173, -114.225, 3.341, 60.906, 41.149] deg
    Waypoint Right_Hole_10: TCP in base x=-289.595 y=723.359 z=43.588 mm, rx=-1.8156 ry=0.6846 rz=-1.8051 rad; joints [140.827, -127.475, -118.143, 4.367, 59.733, 43.565] deg
    Waypoint Right_Hole_11: TCP in base x=-289.905 y=683.248 z=43.271 mm, rx=-1.8157 ry=0.6845 rz=-1.8052 rad; joints [143.448, -125.804, -121.937, 5.097, 58.506, 46.262] deg
  MoveL speed 250 mm/s, acceleration 1200 mm/s^2 (useActiveTCP=true) feature=Base
    Waypoint App_Left: TCP in base x=71.596 y=722.403 z=247.152 mm, rx=1.2411 ry=-1.1842 rz=-1.247 rad; joints [84.654, -103.11, -124.444, -129.739, -95.317, 0.645] deg
  MoveJ speed 60 deg/s, acceleration 80 deg/s^2 (useActiveTCP=true) feature=Center_Left
    Waypoint Left_Hole_1: TCP in base x=41.747 y=681.929 z=288.064 mm, rx=1.241 ry=-1.1844 rz=-1.2467 rad; joints [87.736, -95.501, -128.056, -133.774, -92.257, 0.486] deg; feature pose in base x=41.627 y=722.371 z=247.13 mm, rx=1.2411 ry=-1.1843 rz=-1.2469 rad
    Waypoint Left_hole_2: TCP in base x=41.851 y=761.933 z=289.563 mm, rx=1.241 ry=-1.1846 rz=-1.2468 rad; joints [88.048, -101.94, -119.992, -135.397, -91.927, 0.472] deg
    Waypoint Left_Hole_3: TCP in base x=41.78 y=700.693 z=268.277 mm, rx=1.2407 ry=-1.1848 rz=-1.2467 rad; joints [87.825, -98.689, -127.06, -131.593, -92.143, 0.481] deg
    Waypoint Left_Hole_4: TCP in base x=41.829 y=741.625 z=268.564 mm, rx=1.2407 ry=-1.1848 rz=-1.2468 rad; joints [87.983, -101.916, -122.916, -132.511, -91.98, 0.478] deg
    Waypoint Left_Hole_5: TCP in base x=41.621 y=681.741 z=247.936 mm, rx=1.2407 ry=-1.1848 rz=-1.2466 rad; joints [87.758, -98.951, -129.738, -128.658, -92.209, 0.483] deg
    Waypoint Left_Hole_6: TCP in base x=41.661 y=721.943 z=248.573 mm, rx=1.2412 ry=-1.1844 rz=-1.247 rad; joints [87.923, -102.032, -125.679, -129.603, -92.048, 0.482] deg
    Waypoint Left_Hole_7: TCP in base x=41.655 y=761.751 z=248.951 mm, rx=1.2409 ry=-1.1844 rz=-1.2466 rad; joints [88.067, -105.009, -121.541, -130.787, -91.907, 0.479] deg
    Waypoint Left_Hole_8: TCP in base x=41.551 y=701.515 z=228.336 mm, rx=1.2406 ry=-1.1849 rz=-1.2464 rad; joints [87.856, -102.268, -128.442, -126.647, -92.104, 0.476] deg
    Waypoint Left_Hole_9: TCP in base x=41.634 y=742.006 z=228.723 mm, rx=1.2408 ry=-1.1848 rz=-1.2467 rad; joints [88.007, -105.221, -124.269, -127.852, -91.948, 0.477] deg
    Waypoint Left_Hole_10: TCP in base x=41.475 y=682.374 z=207.743 mm, rx=1.2403 ry=-1.1849 rz=-1.2465 rad; joints [87.783, -102.844, -131.026, -123.494, -92.168, 0.493] deg
    Waypoint Left_Hole_11: TCP in base x=41.584 y=762.28 z=209.041 mm, rx=1.2405 ry=-1.1851 rz=-1.2466 rad; joints [88.087, -108.35, -122.704, -126.306, -91.852, 0.471] deg
SubProgram PickUp (keepSynchronizedWithDisk=false)
  SafeHome (positionOptionType=SPEED_AND_ACCELERATION speed=1.047198 acceleration=1.396263 nextMotionTime=2)
  Set DigitalOutput pin=digital_out[6]; digitalValue=1
  MoveJ speed 60 deg/s, acceleration 80 deg/s^2 (useActiveTCP=true) feature=Base
    Waypoint app_PickUp: TCP in base x=-522.325 y=321.239 z=142.105 mm, rx=1.6368 ry=-0.6237 rz=0.5398 rad; joints [146.504, -113.485, -133.145, 22.41, 109.36, 150.81] deg
  URCap Move Shank (OnRobot, OnRobot A/S) dataModel(or-initialized=true, sd-target-pos=0.035)
    '35mm '
  MoveL speed 250 mm/s, acceleration 1200 mm/s^2 (useActiveTCP=true) feature=Base
    Waypoint Waypoint_1: TCP in base x=-522.33 y=306.822 z=141.634 mm, rx=1.6367 ry=-0.6237 rz=0.5399 rad; joints [147.77, -113.023, -134.336, 23.433, 108.455, 151.739] deg
  Force Frame feature=Center_Pickup; selection=[0, 0, 1, 0, 0, 0]; wrench=[0, 0, 5, 0, 0, 0]; limitsForce=[0.15, 0.15, 0.005, 1.047198, 1.047198, 1.047198]; limitsMotion=[0.1, 0.1, 0.1, 0.349066, 0.349066, 0.349066]
    bOppakken := 1
    Wait Sleep waitTime=4
  Wait Sleep waitTime=0.01
  Set DigitalOutput pin=digital_out[6]; digitalValue=0
  bOppakken := 0
  Script: sd_stop(0)
  Wait Sleep waitTime=0
  MoveL speed 250 mm/s, acceleration 1200 mm/s^2 (useActiveTCP=true) feature=Base
    Waypoint pOmhoogZ (Relative): relativeFromPosition TCP in base x=-522.304 y=306.823 z=141.625 mm, rx=1.6367 ry=-0.6237 rz=0.5399 rad; joints [147.769, -113.023, -134.338, 23.434, 108.455, 151.737] deg; TCP in base x=-522.327 y=306.819 z=171.615 mm, rx=1.6368 ry=-0.6237 rz=0.5399 rad; joints [147.772, -109.464, -133.984, 19.521, 108.459, 151.728] deg
  URCap Move Shank (OnRobot, OnRobot A/S) dataModel(or-initialized=true, sd-target-pos=0.0)
    '35mm '
  Wait Sleep waitTime=1
  Set DigitalOutput pin=digital_out[6]; digitalValue=1
SubProgram Route_Left (keepSynchronizedWithDisk=false)
  MoveJ speed 60 deg/s, acceleration 80 deg/s^2 (useActiveTCP=true) feature=Base
    Waypoint Start_Home: TCP in base x=-422.908 y=487.357 z=157.584 mm, rx=-3.0115 ry=0.7424 rz=0.0187 rad; joints [144.514, -115.165, -138.926, 75.412, 97.807, 88.299] deg
    Waypoint Route_Left1: motionParameters(blendRadius=0.1); TCP in base x=-148.231 y=360.993 z=325.873 mm, rx=-2.2086 ry=0.0374 rz=-2.1865 rad; joints [152.775, -68.83, -133.505, -66.009, 88.321, 62.239] deg
  MoveL speed 250 mm/s, acceleration 1200 mm/s^2 (useActiveTCP=true) feature=Base
    Waypoint Route_Left2: motionParameters(blendRadius=0.1); TCP in base x=229.722 y=360.017 z=324.98 mm, rx=-1.3846 ry=-0.0969 rz=-2.7517 rad; joints [123.932, -57.218, -148.647, -85.145, 59.55, 34.309] deg
  MoveJ speed 60 deg/s, acceleration 80 deg/s^2 (useActiveTCP=true) feature=Base
    Waypoint Route_Left3: motionParameters(blendRadius=0.05); TCP in base x=65.767 y=485.402 z=324.996 mm, rx=1.6131 ry=-0.8684 rz=-1.7053 rad; joints [84.345, -88.18, -152.874, -83.2, -91.449, 3.654] deg
    Waypoint App_Left: TCP in base x=71.596 y=722.403 z=247.152 mm, rx=1.2411 ry=-1.1842 rz=-1.247 rad; joints [84.654, -103.11, -124.444, -129.739, -95.317, 0.645] deg
SubProgram ScrewIn_Left (keepSynchronizedWithDisk=false)
  Wait Sleep waitTime=0.01
  URCap Move Shank (OnRobot, OnRobot A/S) dataModel(or-initialized=true, sd-target-pos=0.035)
    'Add conditions here'
  Script: Postion(Route_Index_1,1 ,arrayStartX,arrayStartZ)
  bIndraaien := 1
  Force Frame feature=Center_Left; selection=[0, 0, 1, 0, 0, 0]; wrench=[0, 0, 2, 0, 0, 0]; limitsForce=[0.15, 0.15, 0.025, 1.047198, 1.047198, 1.047198]; limitsMotion=[0.1, 0.1, 0.1, 0.349066, 0.349066, 0.349066]
    Wait Condition expression=get_sd_Current_torque()>0.5
    Script: sd_stop(0)
  bIndraaien := 0
  Wait Sleep waitTime=0.01
  Script: Postion(Route_Index_1,1 ,arrayFinishX,arrayFinishZ)
  Wait Sleep waitTime=0.01
SubProgram ScrewOut_Left (keepSynchronizedWithDisk=false)
  Force Frame feature=Center_Left; selection=[0, 0, 1, 0, 0, 0]; wrench=[0, 0, -5, 0, 0, 0]; limitsForce=[0.15, 0.15, 0.0025, 1.047198, 1.047198, 1.047198]; limitsMotion=[0.1, 0.1, 0.1, 0.349066, 0.349066, 0.349066]
    URCap Loosen Screw (OnRobot, OnRobot A/S) dataModel(or-initialized=true, sd-length-A=0.035, sd-length-B=0.0)
      'Add conditions here'
  Wait Sleep waitTime=0.01
SubProgram Return_Left (keepSynchronizedWithDisk=false)
  MoveJ speed 60 deg/s, acceleration 80 deg/s^2 (useActiveTCP=true) feature=Base
    Waypoint App_Left: TCP in base x=71.596 y=722.403 z=247.152 mm, rx=1.2411 ry=-1.1842 rz=-1.247 rad; joints [84.654, -103.11, -124.444, -129.739, -95.317, 0.645] deg
    Waypoint Route_Left3: motionParameters(blendRadius=0.05); TCP in base x=65.767 y=485.402 z=324.996 mm, rx=1.6131 ry=-0.8684 rz=-1.7053 rad; joints [84.345, -88.18, -152.874, -83.2, -91.449, 3.654] deg
    Waypoint Route_Left2: motionParameters(blendRadius=0.1); TCP in base x=229.722 y=360.017 z=324.98 mm, rx=-1.3846 ry=-0.0969 rz=-2.7517 rad; joints [123.932, -57.218, -148.647, -85.145, 59.55, 34.309] deg
  MoveL speed 250 mm/s, acceleration 1200 mm/s^2 (useActiveTCP=true) feature=Base
    Waypoint Route_Left1: motionParameters(blendRadius=0.1); TCP in base x=-148.231 y=360.993 z=325.873 mm, rx=-2.2086 ry=0.0374 rz=-2.1865 rad; joints [152.775, -68.83, -133.505, -66.009, 88.321, 62.239] deg
  MoveJ speed 60 deg/s, acceleration 80 deg/s^2 (useActiveTCP=true) feature=Base
    Waypoint Start_Home: TCP in base x=-422.908 y=487.357 z=157.584 mm, rx=-3.0115 ry=0.7424 rz=0.0187 rad; joints [144.514, -115.165, -138.926, 75.412, 97.807, 88.299] deg
SubProgram Route_Slope (keepSynchronizedWithDisk=false)
  MoveJ speed 60 deg/s, acceleration 80 deg/s^2 (useActiveTCP=true) feature=Base
    Waypoint Start_Home: TCP in base x=-422.908 y=487.357 z=157.584 mm, rx=-3.0115 ry=0.7424 rz=0.0187 rad; joints [144.514, -115.165, -138.926, 75.412, 97.807, 88.299] deg
    Waypoint Route_Slope1: motionParameters(blendRadius=0.05); TCP in base x=-469.624 y=632.284 z=161.349 mm, rx=-2.6479 ry=0.7345 rz=-0.8629 rad; joints [144.962, -113.411, -121.258, 26.301, 87.737, 65.268] deg
    Waypoint App_Slope: TCP in base x=-439.97 y=727.052 z=233.948 mm, rx=-1.2131 ry=0.0047 rz=-2.8458 rad; joints [144.347, -130.504, -80.638, -95.321, 64.034, 60.975] deg
SubProgram ScrewIn_Slope (keepSynchronizedWithDisk=false)
  Wait Sleep waitTime=0.01
  URCap Move Shank (OnRobot, OnRobot A/S) dataModel(or-initialized=true, sd-target-pos=0.035)
    'Add conditions here'
  Script: Postion(Route_Index_1,1 ,arrayStartX,arrayStartZ)
  bIndraaien := 1
  Force Frame feature=Center_Slope; selection=[0, 0, 1, 0, 0, 0]; wrench=[0, 0, 2.5, 0, 0, 0]; limitsForce=[0.15, 0.15, 0.03, 1.047198, 1.047198, 1.047198]; limitsMotion=[0.1, 0.1, 0.1, 0.349066, 0.349066, 0.349066]
    Wait Condition expression=get_sd_Current_torque()>0.7
    Script: sd_stop(0)
  Wait Sleep waitTime=0.01
  bIndraaien := 0
  Script: Postion(Route_Index_1,1 ,arrayFinishX,arrayFinishZ)
  Wait Sleep waitTime=0.01
SubProgram ScrewOut_Slope (keepSynchronizedWithDisk=false)
  Force Frame feature=Center_Slope; selection=[0, 0, 1, 0, 0, 0]; wrench=[0, 0, -2.5, 0, 0, 0]; limitsForce=[0.15, 0.15, 0.0025, 1.047198, 1.047198, 1.047198]; limitsMotion=[0.1, 0.1, 0.1, 0.349066, 0.349066, 0.349066]
    URCap Loosen Screw (OnRobot, OnRobot A/S) dataModel(or-initialized=true, sd-length-A=0.035, sd-length-B=0.0)
      'Add conditions here'
  Wait Sleep waitTime=0.01
SubProgram Retrun_Slope (keepSynchronizedWithDisk=false)
  MoveJ speed 60 deg/s, acceleration 80 deg/s^2 (useActiveTCP=true) feature=Base
    Waypoint App_Slope: TCP in base x=-439.97 y=727.052 z=233.948 mm, rx=-1.2131 ry=0.0047 rz=-2.8458 rad; joints [144.347, -130.504, -80.638, -95.321, 64.034, 60.975] deg
    Waypoint Route_Slope1: motionParameters(blendRadius=0.05); TCP in base x=-469.624 y=632.284 z=161.349 mm, rx=-2.6479 ry=0.7345 rz=-0.8629 rad; joints [144.962, -113.411, -121.258, 26.301, 87.737, 65.268] deg
    Waypoint Start_Home: TCP in base x=-422.908 y=487.357 z=157.584 mm, rx=-3.0115 ry=0.7424 rz=0.0187 rad; joints [144.514, -115.165, -138.926, 75.412, 97.807, 88.299] deg
SubProgram Route_Back (keepSynchronizedWithDisk=false)
  MoveJ speed 60 deg/s, acceleration 80 deg/s^2 (useActiveTCP=true) feature=Base
    Waypoint Start_Home: TCP in base x=-422.908 y=487.357 z=157.584 mm, rx=-3.0115 ry=0.7424 rz=0.0187 rad; joints [144.514, -115.165, -138.926, 75.412, 97.807, 88.299] deg
    Waypoint Route_Back1: motionParameters(blendRadius=0.1); TCP in base x=-207.247 y=477.432 z=302.27 mm, rx=-1.9446 ry=0.0025 rz=-1.435 rad; joints [154.944, -69.692, -144.325, -24.25, 78.896, 31.429] deg
    Waypoint App_Back: TCP in base x=-123.1 y=531.725 z=421.395 mm, rx=-1.1912 ry=-1.1756 rz=-1.1726 rad; joints [133.279, -56.474, -130.364, -80.605, 90.835, -48.335] deg
SubProgram ScrewIn_Back (keepSynchronizedWithDisk=false)
  Wait Sleep waitTime=0.01
  URCap Move Shank (OnRobot, OnRobot A/S) dataModel(or-initialized=true, sd-target-pos=0.035)
    'Add conditions here'
  Script: Postion(Route_Index_1,1 ,arrayStartX,arrayStartZ)
  bIndraaien := 1
  Force Frame feature=Center_Back; selection=[0, 0, 1, 0, 0, 0]; wrench=[0, 0, 2, 0, 0, 0]; limitsForce=[0.15, 0.15, 0.025, 1.047198, 1.047198, 1.047198]; limitsMotion=[0.1, 0.1, 0.1, 0.349066, 0.349066, 0.349066]
    Wait Condition expression=get_sd_Current_torque()>0.5
    Script: sd_stop(0)
  Wait Sleep waitTime=0.01
  bIndraaien := 0
  Wait Sleep waitTime=0.01
  Script: Postion(Route_Index_1,1 ,arrayFinishX,arrayFinishZ)
  Wait Sleep waitTime=0.01
SubProgram ScrewOut_Back (keepSynchronizedWithDisk=false)
  Force Frame feature=Center_Back; selection=[0, 0, 1, 0, 0, 0]; wrench=[0, 0, -2.5, 0, 0, 0]; limitsForce=[0.15, 0.15, 0.0025, 1.047198, 1.047198, 1.047198]; limitsMotion=[0.1, 0.1, 0.1, 0.349066, 0.349066, 0.349066]
    URCap Loosen Screw (OnRobot, OnRobot A/S) dataModel(or-initialized=true, sd-length-A=0.035, sd-length-B=0.0)
      'Add conditions here'
  Wait Sleep waitTime=0.01
SubProgram Return_Back (keepSynchronizedWithDisk=false)
  MoveJ speed 60 deg/s, acceleration 80 deg/s^2 (useActiveTCP=true) feature=Base
    Waypoint App_Back: TCP in base x=-123.1 y=531.725 z=421.395 mm, rx=-1.1912 ry=-1.1756 rz=-1.1726 rad; joints [133.279, -56.474, -130.364, -80.605, 90.835, -48.335] deg
    Waypoint Route_Back1: motionParameters(blendRadius=0.1); TCP in base x=-207.247 y=477.432 z=302.27 mm, rx=-1.9446 ry=0.0025 rz=-1.435 rad; joints [154.944, -69.692, -144.325, -24.25, 78.896, 31.429] deg
    Waypoint Start_Home: TCP in base x=-422.908 y=487.357 z=157.584 mm, rx=-3.0115 ry=0.7424 rz=0.0187 rad; joints [144.514, -115.165, -138.926, 75.412, 97.807, 88.299] deg
SubProgram Route_Right (keepSynchronizedWithDisk=false)
  MoveJ speed 60 deg/s, acceleration 80 deg/s^2 (useActiveTCP=true) feature=Base
    Waypoint Start_Home: TCP in base x=-422.908 y=487.357 z=157.584 mm, rx=-3.0115 ry=0.7424 rz=0.0187 rad; joints [144.514, -115.165, -138.926, 75.412, 97.807, 88.299] deg
    Waypoint Route_Right1: motionParameters(blendRadius=0.1); TCP in base x=-469.622 y=632.303 z=80.925 mm, rx=-2.6479 ry=0.7346 rz=-0.8628 rad; joints [144.961, -120.991, -122.125, 34.754, 87.715, 65.278] deg
    Waypoint App_Right: TCP in base x=-319.122 y=726.35 z=84.615 mm, rx=-1.8156 ry=0.6848 rz=-1.8051 rad; joints [142.098, -124.495, -115.917, -1.496, 59.13, 44.861] deg; TCP offset x=153 y=0 z=95.6 mm, rx=0 ry=1.5708 rz=0 rad
SubProgram ScrewIn_Right (keepSynchronizedWithDisk=false)
  URCap Move Shank (OnRobot, OnRobot A/S) dataModel(or-initialized=true, sd-target-pos=0.035)
    'Add conditions here'
  Script: Postion(Route_Index_1,1 ,arrayStartX,arrayStartZ)
  bIndraaien := 1
  Force Frame feature=Center_Right; selection=[0, 0, 1, 0, 0, 0]; wrench=[0, 0, 2, 0, 0, 0]; limitsForce=[0.15, 0.15, 0.025, 1.047198, 1.047198, 1.047198]; limitsMotion=[0.1, 0.1, 0.1, 0.349066, 0.349066, 0.349066]
    Wait Condition expression=get_sd_Current_torque()>0.7
    Script: sd_stop(0)
  bIndraaien := 0
  Script: Postion(Route_Index_1,1 ,arrayFinishX,arrayFinishZ)
  Wait Sleep waitTime=0.01
SubProgram ScrewOut_Right (keepSynchronizedWithDisk=false)
  Force Frame feature=Center_Right; selection=[0, 0, 1, 0, 0, 0]; wrench=[0, 0, 5, 0, 0, 0]; limitsForce=[0.15, 0.15, 0.0025, 1.047198, 1.047198, 1.047198]; limitsMotion=[0.1, 0.1, 0.1, 0.349066, 0.349066, 0.349066]
    URCap Loosen Screw (OnRobot, OnRobot A/S) dataModel(or-initialized=true, sd-length-A=0.035, sd-length-B=0.0)
      'Add conditions here'
  Wait Sleep waitTime=0.01
SubProgram Retrun_Right (keepSynchronizedWithDisk=false)
  MoveJ speed 60 deg/s, acceleration 80 deg/s^2 (useActiveTCP=true) feature=Base
    Waypoint App_Right: TCP in base x=-319.122 y=726.35 z=84.615 mm, rx=-1.8156 ry=0.6848 rz=-1.8051 rad; joints [142.098, -124.495, -115.917, -1.496, 59.13, 44.861] deg
    Waypoint Route_Right1: motionParameters(blendRadius=0.1); TCP in base x=-469.622 y=632.303 z=80.925 mm, rx=-2.6479 ry=0.7346 rz=-0.8628 rad; joints [144.961, -120.991, -122.125, 34.754, 87.715, 65.278] deg; TCP offset x=153 y=0 z=95.6 mm, rx=0 ry=1.5708 rz=0 rad
    Waypoint Start_Home: TCP in base x=-422.908 y=487.357 z=157.584 mm, rx=-3.0115 ry=0.7424 rz=0.0187 rad; joints [144.514, -115.165, -138.926, 75.412, 97.807, 88.299] deg
SubProgram Route_Upside (keepSynchronizedWithDisk=false)
  MoveJ speed 60 deg/s, acceleration 80 deg/s^2 (useActiveTCP=true) feature=Base
    Waypoint Start_Home: TCP in base x=-422.908 y=487.357 z=157.584 mm, rx=-3.0115 ry=0.7424 rz=0.0187 rad; joints [144.514, -115.165, -138.926, 75.412, 97.807, 88.299] deg
    Waypoint Route_Upside1: motionParameters(jointSpeed=1.047198 jointAcceleration=1.396263 cartesianSpeed=0.25 cartesianAcceleration=1.2 blendRadius=0.1); TCP in base x=-148.182 y=360.986 z=325.833 mm, rx=-2.2085 ry=0.0374 rz=-2.1867 rad; joints [152.773, -68.83, -133.51, -66.012, 88.32, 62.236] deg
  MoveL speed 250 mm/s, acceleration 1200 mm/s^2 (useActiveTCP=true) feature=Base
    Waypoint Route_Upside2: motionParameters(blendRadius=0.095); TCP in base x=229.723 y=360.001 z=324.96 mm, rx=-1.3846 ry=-0.097 rz=-2.7518 rad; joints [123.932, -57.218, -148.649, -85.146, 59.552, 34.309] deg
  MoveJ speed 60 deg/s, acceleration 80 deg/s^2 (useActiveTCP=true) feature=Base
    Waypoint Route_Upside3: motionParameters(blendRadius=0.1); TCP in base x=272.03 y=571.295 z=393.795 mm, rx=0.0294 ry=-0.0528 rz=-2.6565 rad; joints [100.801, -96.18, -132.92, -129.415, -17.042, 86.191] deg
    Waypoint App_Upside: TCP in base x=44.432 y=722.092 z=392.585 mm, rx=0.0098 ry=0.0116 rz=-1.5803 rad; joints [105.261, -99.805, -128.74, -130.763, -74.252, 90.052] deg
SubProgram ScrewIn_Upside (keepSynchronizedWithDisk=false)
  Wait Sleep waitTime=0.01
  URCap Move Shank (OnRobot, OnRobot A/S) dataModel(or-initialized=true, sd-target-pos=0.035)
    'Add conditions here'
  Script: Postion(Route_Index_1,1 ,arrayStartX,arrayStartZ)
  bIndraaien := 1
  Force Frame feature=Center_Upside; selection=[0, 0, 1, 0, 0, 0]; wrench=[0, 0, 1.5, 0, 0, 0]; limitsForce=[0.15, 0.15, 0.025, 1.047198, 1.047198, 1.047198]; limitsMotion=[0.1, 0.1, 0.1, 0.349066, 0.349066, 0.349066]
    Wait Condition expression=get_sd_Current_torque()>0.7
    Script: sd_stop(0)
  bIndraaien := 0
  Wait Sleep waitTime=0.01
  Script: Postion(Route_Index_1,1 ,arrayFinishX,arrayFinishZ)
  Wait Sleep waitTime=0.01
SubProgram ScrewOut_Upside (keepSynchronizedWithDisk=false)
  Force Frame feature=Center_Upside; selection=[0, 0, 1, 0, 0, 0]; wrench=[0, 0, -2.5, 0, 0, 0]; limitsForce=[0.15, 0.15, 0.0025, 1.047198, 1.047198, 1.047198]; limitsMotion=[0.1, 0.1, 0.1, 0.349066, 0.349066, 0.349066]
    URCap Loosen Screw (OnRobot, OnRobot A/S) dataModel(or-initialized=true, sd-length-A=0.035, sd-length-B=0.0)
      'Add conditions here'
  Wait Sleep waitTime=0.01
SubProgram Return_Upside (keepSynchronizedWithDisk=false)
  MoveJ speed 60 deg/s, acceleration 80 deg/s^2 (useActiveTCP=true) feature=Base
    Waypoint App_Upside: TCP in base x=44.432 y=722.092 z=392.585 mm, rx=0.0098 ry=0.0116 rz=-1.5803 rad; joints [105.261, -99.805, -128.74, -130.763, -74.252, 90.052] deg
    Waypoint Route_Upside3: motionParameters(blendRadius=0.1); TCP in base x=272.03 y=571.295 z=393.795 mm, rx=0.0294 ry=-0.0528 rz=-2.6565 rad; joints [100.801, -96.18, -132.92, -129.415, -17.042, 86.191] deg
    Waypoint Route_Upside2: TCP in base x=229.723 y=360.001 z=324.96 mm, rx=-1.3846 ry=-0.097 rz=-2.7518 rad; joints [123.932, -57.218, -148.649, -85.146, 59.552, 34.309] deg
  MoveL speed 250 mm/s, acceleration 1200 mm/s^2 (useActiveTCP=true) feature=Base
    Waypoint Route_Upside1: motionParameters(blendRadius=0.1); TCP in base x=-148.182 y=360.986 z=325.833 mm, rx=-2.2085 ry=0.0374 rz=-2.1867 rad; joints [152.773, -68.83, -133.51, -66.012, 88.32, 62.236] deg
  MoveJ speed 60 deg/s, acceleration 80 deg/s^2 (useActiveTCP=true) feature=Base
    Waypoint Start_Home: TCP in base x=-422.908 y=487.357 z=157.584 mm, rx=-3.0115 ry=0.7424 rz=0.0187 rad; joints [144.514, -115.165, -138.926, 75.412, 97.807, 88.299] deg
SubProgram Route_Flat (keepSynchronizedWithDisk=false)
  MoveJ speed 60 deg/s, acceleration 80 deg/s^2 (useActiveTCP=true) feature=Base
    Waypoint Start_Home: TCP in base x=-422.908 y=487.357 z=157.584 mm, rx=-3.0115 ry=0.7424 rz=0.0187 rad; joints [144.514, -115.165, -138.926, 75.412, 97.807, 88.299] deg
    Waypoint Route_Flat1: motionParameters(blendRadius=0.1); TCP in base x=-550.153 y=616.64 z=352.361 mm, rx=-3.0009 ry=0.7398 rz=0.0539 rad; joints [141.481, -107.753, -115.131, 45.664, 100.904, 88.372] deg
    Waypoint App_Flat: TCP in base x=-298.667 y=726.067 z=444.64 mm, rx=-0.093 ry=3.1337 rz=-0.0054 rad; joints [137.032, -122.864, -79.694, 22.109, -43.59, 90.001] deg
SubProgram ScrewIn_Flat (keepSynchronizedWithDisk=false)
  URCap Move Shank (OnRobot, OnRobot A/S) dataModel(or-initialized=true, sd-target-pos=0.035)
    'Add conditions here'
  Script: Postion(Route_Index_1,1 ,arrayStartX,arrayStartZ)
  bIndraaien := 1
  Force Frame feature=Center_Flat; selection=[0, 0, 1, 0, 0, 0]; wrench=[0, 0, 2, 0, 0, 0]; limitsForce=[0.15, 0.15, 0.025, 1.047198, 1.047198, 1.047198]; limitsMotion=[0.1, 0.1, 0.1, 0.349066, 0.349066, 0.349066]
    Wait Condition expression=get_sd_Current_torque()>0.5
    Script: sd_stop(0)
  bIndraaien := 0
  Script: Postion(Route_Index_1,1 ,arrayFinishX,arrayFinishZ)
  Wait Sleep waitTime=0.01
SubProgram ScrewOut_Flat (keepSynchronizedWithDisk=false)
  Force Frame feature=Center_Flat; selection=[0, 0, 1, 0, 0, 0]; wrench=[0, 0, -2.5, 0, 0, 0]; limitsForce=[0.15, 0.15, 0.0045, 1.047198, 1.047198, 1.047198]; limitsMotion=[0.1, 0.1, 0.1, 0.349066, 0.349066, 0.349066]
    URCap Loosen Screw (OnRobot, OnRobot A/S) dataModel(or-initialized=true, sd-length-A=0.035, sd-length-B=0.001)
      'Add conditions here'
  Wait Sleep waitTime=0.01
SubProgram Return_Flat (keepSynchronizedWithDisk=false)
  MoveJ speed 60 deg/s, acceleration 80 deg/s^2 (useActiveTCP=true) feature=Base
    Waypoint App_Flat: TCP in base x=-298.667 y=726.067 z=444.64 mm, rx=-0.093 ry=3.1337 rz=-0.0054 rad; joints [137.032, -122.864, -79.694, 22.109, -43.59, 90.001] deg
    Waypoint Route_Flat1: motionParameters(blendRadius=0.1); TCP in base x=-550.153 y=616.64 z=352.361 mm, rx=-3.0009 ry=0.7398 rz=0.0539 rad; joints [141.481, -107.753, -115.131, 45.664, 100.904, 88.372] deg
    Waypoint Start_Home: TCP in base x=-422.908 y=487.357 z=157.584 mm, rx=-3.0115 ry=0.7424 rz=0.0187 rad; joints [144.514, -115.165, -138.926, 75.412, 97.807, 88.299] deg
